	VAR robtarget Openhole_6212 := [[422.92, 1.19, 186.57], [-0.151917, 0.690595, 0.706732, 0.02301], [0,0,0,0], [9E9, 9E9, 9E9, 9E9, 9E9, 9E9]];
	VAR robtarget Openhole_6213 := [[423.41, 1.3, 186.5], [-0.15063, 0.690877, 0.706788, 0.021231], [0,0,0,0], [9E9, 9E9, 9E9, 9E9, 9E9, 9E9]];
	VAR robtarget Openhole_6214 := [[417.57, 1.3, 187.64], [-0.167714, 0.686929, 0.705941, 0.040584], [0,0,0,0], [9E9, 9E9, 9E9, 9E9, 9E9, 9E9]];
	VAR robtarget Openhole_6215 := [[417.07, 1.15, 187.69], [-0.168902, 0.686638, 0.705835, 0.042396], [0,0,0,0], [9E9, 9E9, 9E9, 9E9, 9E9, 9E9]];
	VAR robtarget Openhole_6216 := [[408.73, 0.11, 188.91], [-0.188817, 0.681431, 0.703403, 0.072276], [0,0,0,0], [9E9, 9E9, 9E9, 9E9, 9E9, 9E9]];
	VAR robtarget Openhole_6217 := [[397.88, -0.81, 190.45], [-0.213744, 0.674028, 0.698859, 0.107688], [0,0,0,0], [9E9, 9E9, 9E9, 9E9, 9E9, 9E9]];
	VAR robtarget Openhole_6218 := [[394.38, -1.04, 190.94], [-0.221411, 0.671548, 0.697131, 0.118354], [0,0,0,0], [9E9, 9E9, 9E9, 9E9, 9E9, 9E9]];
	VAR robtarget Openhole_6219 := [[389.38, -1.04, 191.81], [-0.232781, 0.667692, 0.694645, 0.13217], [0,0,0,0], [9E9, 9E9, 9E9, 9E9, 9E9, 9E9]];
	VAR robtarget Openhole_6220 := [[362.42, -1.04, 191.89], [-0.183051, 0.683002, 0.683002, 0.183051], [0,0,0,0], [9E9, 9E9, 9E9, 9E9, 9E9, 9E9]];
	VAR robtarget Openhole_6221 := [[362.42, -1.04, 192.01], [-0.183051, 0.683002, 0.683002, 0.183051], [0,0,0,0], [9E9, 9E9, 9E9, 9E9, 9E9, 9E9]];
	VAR robtarget Openhole_6222 := [[389.38, -1.04, 191.93], [-0.232953, 0.667632, 0.694664, 0.132066], [0,0,0,0], [9E9, 9E9, 9E9, 9E9, 9E9, 9E9]];
	VAR robtarget Openhole_6223 := [[394.38, -1.04, 191.06], [-0.221583, 0.671492, 0.697148, 0.118257], [0,0,0,0], [9E9, 9E9, 9E9, 9E9, 9E9, 9E9]];
	VAR robtarget Openhole_6224 := [[406.26, -0.14, 189.38], [-0.194769, 0.679754, 0.702502, 0.080567], [0,0,0,0], [9E9, 9E9, 9E9, 9E9, 9E9, 9E9]];
	VAR robtarget Openhole_6225 := [[415.12, 0.87, 188.1], [-0.173761, 0.685425, 0.705366, 0.049587], [0,0,0,0], [9E9, 9E9, 9E9, 9E9, 9E9, 9E9]];
	VAR robtarget Openhole_6226 := [[417.07, 1.15, 187.81], [-0.16906, 0.686599, 0.705837, 0.042358], [0,0,0,0], [9E9, 9E9, 9E9, 9E9, 9E9, 9E9]];
	VAR robtarget Openhole_6227 := [[417.57, 1.3, 187.76], [-0.167777, 0.686914, 0.705937, 0.040655], [0,0,0,0], [9E9, 9E9, 9E9, 9E9, 9E9, 9E9]];
	VAR robtarget Openhole_6228 := [[423.41, 1.3, 186.62], [-0.150696, 0.690862, 0.706786, 0.021304], [0,0,0,0], [9E9, 9E9, 9E9, 9E9, 9E9, 9E9]];
	VAR robtarget Openhole_6229 := [[422.92, 1.19, 186.69], [-0.152065, 0.690562, 0.706733, 0.02299], [0,0,0,0], [9E9, 9E9, 9E9, 9E9, 9E9, 9E9]];
	VAR robtarget Openhole_6230 := [[416.08, 0.05, 187.65], [-0.168515, 0.686733, 0.705405, 0.049029], [0,0,0,0], [9E9, 9E9, 9E9, 9E9, 9E9, 9E9]];
	VAR robtarget Openhole_6231 := [[407.72, -0.93, 188.8], [-0.188593, 0.681493, 0.702735, 0.078506], [0,0,0,0], [9E9, 9E9, 9E9, 9E9, 9E9, 9E9]];
	VAR robtarget Openhole_6232 := [[395.86, -1.84, 190.4], [-0.215851, 0.673356, 0.697466, 0.116368], [0,0,0,0], [9E9, 9E9, 9E9, 9E9, 9E9, 9E9]];
	VAR robtarget Openhole_6233 := [[394.38, -1.93, 190.59], [-0.219087, 0.67231, 0.696705, 0.120837], [0,0,0,0], [9E9, 9E9, 9E9, 9E9, 9E9, 9E9]];
	VAR robtarget Openhole_6234 := [[389.38, -1.93, 191.41], [-0.23052, 0.668476, 0.69418, 0.134588], [0,0,0,0], [9E9, 9E9, 9E9, 9E9, 9E9, 9E9]];
	VAR robtarget Openhole_6235 := [[362.38, -1.93, 191.5], [-0.183051, 0.683002, 0.683002, 0.183051], [0,0,0,0], [9E9, 9E9, 9E9, 9E9, 9E9, 9E9]];
	VAR robtarget Openhole_6236 := [[362.38, -2.82, 190.99], [-0.183051, 0.683002, 0.683002, 0.183051], [0,0,0,0], [9E9, 9E9, 9E9, 9E9, 9E9, 9E9]];
	VAR robtarget Openhole_6237 := [[374.38, -2.82, 190.95], [-0.183051, 0.683002, 0.683002, 0.183051], [0,0,0,0], [9E9, 9E9, 9E9, 9E9, 9E9, 9E9]];
	VAR robtarget Openhole_6238 := [[389.38, -2.82, 190.9], [-0.228098, 0.669306, 0.69369, 0.137092], [0,0,0,0], [9E9, 9E9, 9E9, 9E9, 9E9, 9E9]];
	VAR robtarget Openhole_6239 := [[394.37, -2.82, 190.12], [-0.21661, 0.673112, 0.696255, 0.123408], [0,0,0,0], [9E9, 9E9, 9E9, 9E9, 9E9, 9E9]];
	VAR robtarget Openhole_6240 := [[408.22, -1.78, 188.37], [-0.184687, 0.682562, 0.702618, 0.079551], [0,0,0,0], [9E9, 9E9, 9E9, 9E9, 9E9, 9E9]];
	VAR robtarget Openhole_6241 := [[416.11, -0.88, 187.35], [-0.165576, 0.687448, 0.705202, 0.05187], [0,0,0,0], [9E9, 9E9, 9E9, 9E9, 9E9, 9E9]];
	VAR robtarget Openhole_6242 := [[422.96, 0.24, 186.44], [-0.148993, 0.691232, 0.706633, 0.025886], [0,0,0,0], [9E9, 9E9, 9E9, 9E9, 9E9, 9E9]];
	VAR robtarget Openhole_6243 := [[427.32, 1.15, 185.82], [-0.138588, 0.693393, 0.707057, 0.008368], [0,0,0,0], [9E9, 9E9, 9E9, 9E9, 9E9, 9E9]];
	VAR robtarget Openhole_6244 := [[427.8, 1.3, 185.76], [-0.137346, 0.69364, 0.707077, 0.006493], [0,0,0,0], [9E9, 9E9, 9E9, 9E9, 9E9, 9E9]];
	VAR robtarget Openhole_6245 := [[431.7, 1.3, 185], [-0.125184, 0.695937, 0.707074, -0.006768], [0,0,0,0], [9E9, 9E9, 9E9, 9E9, 9E9, 9E9]];
	VAR robtarget Openhole_6246 := [[431.22, 1.07, 185.05], [-0.126171, 0.695759, 0.707092, -0.004584], [0,0,0,0], [9E9, 9E9, 9E9, 9E9, 9E9, 9E9]];
	VAR robtarget Openhole_6247 := [[423.97, -0.54, 186.06], [-0.143494, 0.692394, 0.706664, 0.025018], [0,0,0,0], [9E9, 9E9, 9E9, 9E9, 9E9, 9E9]];
	VAR robtarget Openhole_6248 := [[417.11, -1.69, 186.92], [-0.160194, 0.688722, 0.705255, 0.051147], [0,0,0,0], [9E9, 9E9, 9E9, 9E9, 9E9, 9E9]];
	VAR robtarget Openhole_6249 := [[409.23, -2.6, 187.89], [-0.179528, 0.683937, 0.702684, 0.078962], [0,0,0,0], [9E9, 9E9, 9E9, 9E9, 9E9, 9E9]];
	VAR robtarget Openhole_6250 := [[394.87, -3.67, 189.6], [-0.213029, 0.674254, 0.696063, 0.124485], [0,0,0,0], [9E9, 9E9, 9E9, 9E9, 9E9, 9E9]];
	VAR robtarget Openhole_6251 := [[394.37, -3.7, 189.65], [-0.214125, 0.673907, 0.695793, 0.125983], [0,0,0,0], [9E9, 9E9, 9E9, 9E9, 9E9, 9E9]];
	VAR robtarget Openhole_6252 := [[389.37, -3.7, 190.39], [-0.225669, 0.670129, 0.69319, 0.1396], [0,0,0,0], [9E9, 9E9, 9E9, 9E9, 9E9, 9E9]];
	VAR robtarget Openhole_6253 := [[362.37, -3.7, 190.48], [-0.183051, 0.683002, 0.683002, 0.183051], [0,0,0,0], [9E9, 9E9, 9E9, 9E9, 9E9, 9E9]];
	VAR robtarget Openhole_6254 := [[362.37, -4.58, 189.97], [-0.183051, 0.683002, 0.683002, 0.183051], [0,0,0,0], [9E9, 9E9, 9E9, 9E9, 9E9, 9E9]];
	VAR robtarget Openhole_6255 := [[374.37, -4.58, 189.93], [-0.183051, 0.683002, 0.683002, 0.183051], [0,0,0,0], [9E9, 9E9, 9E9, 9E9, 9E9, 9E9]];
	VAR robtarget Openhole_6256 := [[389.37, -4.59, 189.88], [-0.223232, 0.670945, 0.692679, 0.142111], [0,0,0,0], [9E9, 9E9, 9E9, 9E9, 9E9, 9E9]];
	VAR robtarget Openhole_6257 := [[394.36, -4.59, 189.19], [-0.211638, 0.674692, 0.69532, 0.128569], [0,0,0,0], [9E9, 9E9, 9E9, 9E9, 9E9, 9E9]];
	VAR robtarget Openhole_6258 := [[409.74, -3.48, 187.47], [-0.175466, 0.68499, 0.702554, 0.080113], [0,0,0,0], [9E9, 9E9, 9E9, 9E9, 9E9, 9E9]];
	VAR robtarget Openhole_6259 := [[417.63, -2.6, 186.56], [-0.155846, 0.689719, 0.705166, 0.052359], [0,0,0,0], [9E9, 9E9, 9E9, 9E9, 9E9, 9E9]];
	VAR robtarget Openhole_6260 := [[424, -1.56, 185.8], [-0.140137, 0.693081, 0.706546, 0.028167], [0,0,0,0], [9E9, 9E9, 9E9, 9E9, 9E9, 9E9]];
	VAR robtarget Openhole_6261 := [[430.79, -0.09, 184.92], [-0.123778, 0.696189, 0.707106, 0.000643], [0,0,0,0], [9E9, 9E9, 9E9, 9E9, 9E9, 9E9]];
	VAR robtarget Openhole_6262 := [[435.6, 1.08, 184.2], [-0.112198, 0.698149, 0.706837, -0.019526], [0,0,0,0], [9E9, 9E9, 9E9, 9E9, 9E9, 9E9]];
	VAR robtarget Openhole_6263 := [[436.08, 1.3, 184.14], [-0.111001, 0.69834, 0.706766, -0.021958], [0,0,0,0], [9E9, 9E9, 9E9, 9E9, 9E9, 9E9]];
	VAR robtarget Openhole_6264 := [[440.9, 1.3, 183.19], [-0.095242, 0.700663, 0.706058, -0.038495], [0,0,0,0], [9E9, 9E9, 9E9, 9E9, 9E9, 9E9]];
	VAR robtarget Openhole_6265 := [[440.43, 1.14, 183.27], [-0.096594, 0.700478, 0.706178, -0.03623], [0,0,0,0], [9E9, 9E9, 9E9, 9E9, 9E9, 9E9]];
	VAR robtarget Openhole_6266 := [[431.79, -1.04, 184.58], [-0.117568, 0.697265, 0.707107, 0.000299], [0,0,0,0], [9E9, 9E9, 9E9, 9E9, 9E9, 9E9]];
	VAR robtarget Openhole_6267 := [[425, -2.5, 185.42], [-0.134117, 0.694271, 0.706557, 0.027869], [0,0,0,0], [9E9, 9E9, 9E9, 9E9, 9E9, 9E9]];
	VAR robtarget Openhole_6268 := [[418.62, -3.5, 186.14], [-0.150147, 0.690982, 0.705191, 0.052021], [0,0,0,0], [9E9, 9E9, 9E9, 9E9, 9E9, 9E9]];
	VAR robtarget Openhole_6269 := [[410.22, -4.4, 187.05], [-0.171369, 0.686027, 0.702401, 0.081442], [0,0,0,0], [9E9, 9E9, 9E9, 9E9, 9E9, 9E9]];
	VAR robtarget Openhole_6270 := [[394.37, -5.47, 188.72], [-0.209106, 0.675481, 0.694846, 0.131109], [0,0,0,0], [9E9, 9E9, 9E9, 9E9, 9E9, 9E9]];
	VAR robtarget Openhole_6271 := [[389.37, -5.47, 189.37], [-0.22079, 0.671753, 0.692159, 0.144623], [0,0,0,0], [9E9, 9E9, 9E9, 9E9, 9E9, 9E9]];
	VAR robtarget Openhole_6272 := [[362.37, -5.47, 189.46], [-0.183051, 0.683002, 0.683002, 0.183051], [0,0,0,0], [9E9, 9E9, 9E9, 9E9, 9E9, 9E9]];
	VAR robtarget Openhole_6273 := [[362.37, -6.37, 188.93], [-0.183051, 0.683002, 0.683002, 0.183051], [0,0,0,0], [9E9, 9E9, 9E9, 9E9, 9E9, 9E9]];
	VAR robtarget Openhole_6274 := [[374.37, -6.37, 188.9], [-0.183051, 0.683002, 0.683002, 0.183051], [0,0,0,0], [9E9, 9E9, 9E9, 9E9, 9E9, 9E9]];
	VAR robtarget Openhole_6275 := [[389.37, -6.37, 188.85], [-0.21828, 0.672572, 0.691616, 0.147199], [0,0,0,0], [9E9, 9E9, 9E9, 9E9, 9E9, 9E9]];
	VAR robtarget Openhole_6276 := [[394.35, -6.37, 188.24], [-0.206567, 0.676262, 0.694335, 0.133787], [0,0,0,0], [9E9, 9E9, 9E9, 9E9, 9E9, 9E9]];
	VAR robtarget Openhole_6277 := [[411.75, -5.23, 186.54], [-0.164547, 0.687695, 0.702646, 0.079304], [0,0,0,0], [9E9, 9E9, 9E9, 9E9, 9E9, 9E9]];
	VAR robtarget Openhole_6278 := [[420.16, -4.36, 185.66], [-0.142875, 0.692522, 0.705352, 0.049787], [0,0,0,0], [9E9, 9E9, 9E9, 9E9, 9E9, 9E9]];
	VAR robtarget Openhole_6279 := [[427.03, -3.3, 184.92], [-0.125272, 0.695922, 0.70671, 0.023676], [0,0,0,0], [9E9, 9E9, 9E9, 9E9, 9E9, 9E9]];
	VAR robtarget Openhole_6280 := [[432.87, -2.08, 184.23], [-0.110768, 0.698377, 0.707107, 0.000055], [0,0,0,0], [9E9, 9E9, 9E9, 9E9, 9E9, 9E9]];
	VAR robtarget Openhole_6281 := [[441.01, 0.05, 183.07], [-0.091101, 0.701214, 0.706256, -0.034673], [0,0,0,0], [9E9, 9E9, 9E9, 9E9, 9E9, 9E9]];
	VAR robtarget Openhole_6282 := [[444.81, 1.13, 182.42], [-0.081961, 0.702341, 0.705254, -0.051157], [0,0,0,0], [9E9, 9E9, 9E9, 9E9, 9E9, 9E9]];
	VAR robtarget Openhole_6283 := [[445.28, 1.3, 182.34], [-0.080875, 0.702467, 0.705097, -0.053269], [0,0,0,0], [9E9, 9E9, 9E9, 9E9, 9E9, 9E9]];
	VAR robtarget Openhole_6284 := [[492.93, 1.3, 173.01], [0.078403, 0.702747, 0.678324, -0.199693], [0,0,0,0], [9E9, 9E9, 9E9, 9E9, 9E9, 9E9]];
	VAR robtarget Openhole_6285 := [[497.82, 0.35, 172.5], [0.096043, 0.700554, 0.675427, -0.209279], [0,0,0,0], [9E9, 9E9, 9E9, 9E9, 9E9, 9E9]];
	VAR robtarget Openhole_6286 := [[502.17, -0.75, 172.24], [0.112029, 0.698176, 0.673078, -0.216717], [0,0,0,0], [9E9, 9E9, 9E9, 9E9, 9E9, 9E9]];
	VAR robtarget Openhole_6287 := [[503.61, -1.18, 172.21], [0.117389, 0.697295, 0.67237, -0.218903], [0,0,0,0], [9E9, 9E9, 9E9, 9E9, 9E9, 9E9]];
	VAR robtarget Openhole_6288 := [[504.32, -1.34, 172.18], [0.119865, 0.696873, 0.671974, -0.220115], [0,0,0,0], [9E9, 9E9, 9E9, 9E9, 9E9, 9E9]];
	VAR robtarget Openhole_6289 := [[509.32, -1.34, 171.33], [0.183051, 0.683002, 0.683002, -0.183051], [0,0,0,0], [9E9, 9E9, 9E9, 9E9, 9E9, 9E9]];
	VAR robtarget Openhole_6290 := [[536.31, -1.34, 171.24], [0.183051, 0.683002, 0.683002, -0.183051], [0,0,0,0], [9E9, 9E9, 9E9, 9E9, 9E9, 9E9]];
	VAR robtarget Openhole_6291 := [[536.32, -1.86, 171.55], [0.183051, 0.683002, 0.683002, -0.183051], [0,0,0,0], [9E9, 9E9, 9E9, 9E9, 9E9, 9E9]];
	VAR robtarget Openhole_6292 := [[509.32, -1.86, 171.63], [0.183051, 0.683002, 0.683002, -0.183051], [0,0,0,0], [9E9, 9E9, 9E9, 9E9, 9E9, 9E9]];
	VAR robtarget Openhole_6293 := [[504.32, -1.86, 172.46], [0.121395, 0.696608, 0.672454, -0.218646], [0,0,0,0], [9E9, 9E9, 9E9, 9E9, 9E9, 9E9]];
	VAR robtarget Openhole_6294 := [[503.45, -1.68, 172.5], [0.118397, 0.697124, 0.672944, -0.217131], [0,0,0,0], [9E9, 9E9, 9E9, 9E9, 9E9, 9E9]];
	VAR robtarget Openhole_6295 := [[502.98, -1.51, 172.5], [0.116581, 0.69743, 0.673158, -0.216468], [0,0,0,0], [9E9, 9E9, 9E9, 9E9, 9E9, 9E9]];
	VAR robtarget Openhole_6296 := [[498.64, -0.34, 172.67], [0.100548, 0.699922, 0.675418, -0.20931], [0,0,0,0], [9E9, 9E9, 9E9, 9E9, 9E9, 9E9]];
	VAR robtarget Openhole_6297 := [[493.76, 0.68, 173.11], [0.082837, 0.702238, 0.678231, -0.200005], [0,0,0,0], [9E9, 9E9, 9E9, 9E9, 9E9, 9E9]];
	VAR robtarget Openhole_6298 := [[490.83, 1.18, 173.47], [0.07224, 0.703407, 0.680018, -0.193843], [0,0,0,0], [9E9, 9E9, 9E9, 9E9, 9E9, 9E9]];
	VAR robtarget Openhole_6299 := [[490.33, 1.3, 173.52], [0.07032, 0.703601, 0.680285, -0.192906], [0,0,0,0], [9E9, 9E9, 9E9, 9E9, 9E9, 9E9]];
	VAR robtarget Openhole_6300 := [[480.37, 1.3, 175.47], [0.038288, 0.706069, 0.68749, -0.1654], [0,0,0,0], [9E9, 9E9, 9E9, 9E9, 9E9, 9E9]];
	VAR robtarget Openhole_6301 := [[486.27, 0.75, 174.51], [0.059128, 0.70463, 0.683728, -0.180323], [0,0,0,0], [9E9, 9E9, 9E9, 9E9, 9E9, 9E9]];
	VAR robtarget Openhole_6302 := [[492.16, -0.08, 173.73], [0.080181, 0.702546, 0.680077, -0.193637], [0,0,0,0], [9E9, 9E9, 9E9, 9E9, 9E9, 9E9]];
	VAR robtarget Openhole_6303 := [[497.54, -1.09, 173.22], [0.099523, 0.700068, 0.676913, -0.204423], [0,0,0,0], [9E9, 9E9, 9E9, 9E9, 9E9, 9E9]];
	VAR robtarget Openhole_6304 := [[502.87, -2.42, 172.98], [0.118916, 0.697036, 0.674059, -0.213647], [0,0,0,0], [9E9, 9E9, 9E9, 9E9, 9E9, 9E9]];
	VAR robtarget Openhole_6305 := [[503.83, -2.67, 172.96], [0.122383, 0.696436, 0.673553, -0.215236], [0,0,0,0], [9E9, 9E9, 9E9, 9E9, 9E9, 9E9]];
	VAR robtarget Openhole_6306 := [[504.4, -2.79, 172.93], [0.124334, 0.69609, 0.67323, -0.216245], [0,0,0,0], [9E9, 9E9, 9E9, 9E9, 9E9, 9E9]];
	VAR robtarget Openhole_6307 := [[509.32, -2.79, 172.17], [0.183051, 0.683002, 0.683002, -0.183051], [0,0,0,0], [9E9, 9E9, 9E9, 9E9, 9E9, 9E9]];
	VAR robtarget Openhole_6308 := [[536.32, -2.79, 172.08], [0.183051, 0.683002, 0.683002, -0.183051], [0,0,0,0], [9E9, 9E9, 9E9, 9E9, 9E9, 9E9]];
	VAR robtarget Openhole_6309 := [[536.32, -3.66, 172.58], [0.183051, 0.683002, 0.683002, -0.183051], [0,0,0,0], [9E9, 9E9, 9E9, 9E9, 9E9, 9E9]];
	VAR robtarget Openhole_6310 := [[509.32, -3.66, 172.67], [0.183051, 0.683002, 0.683002, -0.183051], [0,0,0,0], [9E9, 9E9, 9E9, 9E9, 9E9, 9E9]];
	VAR robtarget Openhole_6311 := [[504.32, -3.66, 173.41], [0.12664, 0.695674, 0.674075, -0.213596], [0,0,0,0], [9E9, 9E9, 9E9, 9E9, 9E9, 9E9]];
	VAR robtarget Openhole_6312 := [[503.61, -3.55, 173.45], [0.124315, 0.696093, 0.674503, -0.21224], [0,0,0,0], [9E9, 9E9, 9E9, 9E9, 9E9, 9E9]];
	VAR robtarget Openhole_6313 := [[496.78, -2.08, 173.8], [0.100233, 0.699967, 0.678334, -0.199656], [0,0,0,0], [9E9, 9E9, 9E9, 9E9, 9E9, 9E9]];
	VAR robtarget Openhole_6314 := [[490.89, -1.1, 174.37], [0.079383, 0.702637, 0.681857, -0.187272], [0,0,0,0], [9E9, 9E9, 9E9, 9E9, 9E9, 9E9]];
	VAR robtarget Openhole_6315 := [[484.49, -0.34, 175.22], [0.056846, 0.704818, 0.685848, -0.172081], [0,0,0,0], [9E9, 9E9, 9E9, 9E9, 9E9, 9E9]];
	VAR robtarget Openhole_6316 := [[478.08, 0.04, 176.26], [0.034733, 0.706253, 0.689935, -0.154887], [0,0,0,0], [9E9, 9E9, 9E9, 9E9, 9E9, 9E9]];
	VAR robtarget Openhole_6317 := [[475.62, 0.08, 176.71], [0.02643, 0.706613, 0.691506, -0.147712], [0,0,0,0], [9E9, 9E9, 9E9, 9E9, 9E9, 9E9]];
	VAR robtarget Openhole_6318 := [[475.13, 0.08, 176.8], [0.02479, 0.706672, 0.691821, -0.146234], [0,0,0,0], [9E9, 9E9, 9E9, 9E9, 9E9, 9E9]];
	VAR robtarget Openhole_6319 := [[468.75, -0.12, 178.01], [0.00393, 0.707096, 0.69579, -0.126002], [0,0,0,0], [9E9, 9E9, 9E9, 9E9, 9E9, 9E9]];
	VAR robtarget Openhole_6320 := [[461.39, -0.49, 179.39], [-0.020021, 0.706823, 0.699814, -0.101296], [0,0,0,0], [9E9, 9E9, 9E9, 9E9, 9E9, 9E9]];
	VAR robtarget Openhole_6321 := [[460.9, -0.5, 179.48], [-0.021687, 0.706774, 0.700047, -0.099671], [0,0,0,0], [9E9, 9E9, 9E9, 9E9, 9E9, 9E9]];
	VAR robtarget Openhole_6322 := [[459.91, -0.49, 179.66], [-0.025088, 0.706662, 0.700494, -0.096476], [0,0,0,0], [9E9, 9E9, 9E9, 9E9, 9E9, 9E9]];
	VAR robtarget Openhole_6323 := [[457.95, -0.41, 180], [-0.032126, 0.706377, 0.701319, -0.090283], [0,0,0,0], [9E9, 9E9, 9E9, 9E9, 9E9, 9E9]];
	VAR robtarget Openhole_6324 := [[456.96, -0.33, 180.17], [-0.035756, 0.706202, 0.701698, -0.087291], [0,0,0,0], [9E9, 9E9, 9E9, 9E9, 9E9, 9E9]];
	VAR robtarget Openhole_6325 := [[455.49, -0.16, 180.42], [-0.041344, 0.705897, 0.702224, -0.082958], [0,0,0,0], [9E9, 9E9, 9E9, 9E9, 9E9, 9E9]];
	VAR robtarget Openhole_6326 := [[454.52, -0.01, 180.59], [-0.045187, 0.705661, 0.702542, -0.080213], [0,0,0,0], [9E9, 9E9, 9E9, 9E9, 9E9, 9E9]];
	VAR robtarget Openhole_6327 := [[453.56, 0.19, 180.76], [-0.049153, 0.705396, 0.702831, -0.077642], [0,0,0,0], [9E9, 9E9, 9E9, 9E9, 9E9, 9E9]];
	VAR robtarget Openhole_6328 := [[453.08, 0.32, 180.85], [-0.05122, 0.705249, 0.702957, -0.076494], [0,0,0,0], [9E9, 9E9, 9E9, 9E9, 9E9, 9E9]];
	VAR robtarget Openhole_6329 := [[451.65, 0.69, 181.1], [-0.057308, 0.704781, 0.703342, -0.072869], [0,0,0,0], [9E9, 9E9, 9E9, 9E9, 9E9, 9E9]];
	VAR robtarget Openhole_6330 := [[451.17, 0.77, 181.19], [-0.059249, 0.70462, 0.70348, -0.071529], [0,0,0,0], [9E9, 9E9, 9E9, 9E9, 9E9, 9E9]];
	VAR robtarget Openhole_6331 := [[450.68, 0.85, 181.29], [-0.061142, 0.704458, 0.703621, -0.070123], [0,0,0,0], [9E9, 9E9, 9E9, 9E9, 9E9, 9E9]];
	VAR robtarget Openhole_6332 := [[450.19, 0.88, 181.38], [-0.062918, 0.704302, 0.703774, -0.068577], [0,0,0,0], [9E9, 9E9, 9E9, 9E9, 9E9, 9E9]];
	VAR robtarget Openhole_6333 := [[449.7, 0.9, 181.47], [-0.064666, 0.704144, 0.703926, -0.066997], [0,0,0,0], [9E9, 9E9, 9E9, 9E9, 9E9, 9E9]];
	VAR robtarget Openhole_6334 := [[449.21, 0.87, 181.57], [-0.066224, 0.703999, 0.704091, -0.065232], [0,0,0,0], [9E9, 9E9, 9E9, 9E9, 9E9, 9E9]];
	VAR robtarget Openhole_6335 := [[448.72, 0.81, 181.66], [-0.067701, 0.703858, 0.704259, -0.063401], [0,0,0,0], [9E9, 9E9, 9E9, 9E9, 9E9, 9E9]];
	VAR robtarget Openhole_6336 := [[447.76, 0.61, 181.84], [-0.070294, 0.703604, 0.704601, -0.059475], [0,0,0,0], [9E9, 9E9, 9E9, 9E9, 9E9, 9E9]];
	VAR robtarget Openhole_6337 := [[446.81, 0.36, 182.02], [-0.072697, 0.70336, 0.704931, -0.055424], [0,0,0,0], [9E9, 9E9, 9E9, 9E9, 9E9, 9E9]];
	VAR robtarget Openhole_6338 := [[438.73, -1.98, 183.28], [-0.091999, 0.701096, 0.706817, -0.020235], [0,0,0,0], [9E9, 9E9, 9E9, 9E9, 9E9, 9E9]];
	VAR robtarget Openhole_6339 := [[433.44, -3.29, 183.95], [-0.10498, 0.69927, 0.707104, 0.002105], [0,0,0,0], [9E9, 9E9, 9E9, 9E9, 9E9, 9E9]];
	VAR robtarget Openhole_6340 := [[427.09, -4.48, 184.66], [-0.121297, 0.696625, 0.706578, 0.027349], [0,0,0,0], [9E9, 9E9, 9E9, 9E9, 9E9, 9E9]];
	VAR robtarget Openhole_6341 := [[419.69, -5.48, 185.41], [-0.140734, 0.69296, 0.704975, 0.054865], [0,0,0,0], [9E9, 9E9, 9E9, 9E9, 9E9, 9E9]];
	VAR robtarget Openhole_6342 := [[409.78, -6.33, 186.38], [-0.16668, 0.687181, 0.701508, 0.088809], [0,0,0,0], [9E9, 9E9, 9E9, 9E9, 9E9, 9E9]];
	VAR robtarget Openhole_6343 := [[394.35, -7.26, 187.77], [-0.204053, 0.677025, 0.693832, 0.136373], [0,0,0,0], [9E9, 9E9, 9E9, 9E9, 9E9, 9E9]];
	VAR robtarget Openhole_6344 := [[389.37, -7.26, 188.34], [-0.215823, 0.673365, 0.691075, 0.149715], [0,0,0,0], [9E9, 9E9, 9E9, 9E9, 9E9, 9E9]];
	VAR robtarget Openhole_6345 := [[362.37, -7.26, 188.42], [-0.183051, 0.683002, 0.683002, 0.183051], [0,0,0,0], [9E9, 9E9, 9E9, 9E9, 9E9, 9E9]];
	VAR robtarget Openhole_6346 := [[362.37, -8.14, 187.91], [-0.183051, 0.683002, 0.683002, 0.183051], [0,0,0,0], [9E9, 9E9, 9E9, 9E9, 9E9, 9E9]];
	VAR robtarget Openhole_6347 := [[374.37, -8.14, 187.88], [-0.183051, 0.683002, 0.683002, 0.183051], [0,0,0,0], [9E9, 9E9, 9E9, 9E9, 9E9, 9E9]];
	VAR robtarget Openhole_6348 := [[389.37, -8.14, 187.83], [-0.21336, 0.674149, 0.690525, 0.152233], [0,0,0,0], [9E9, 9E9, 9E9, 9E9, 9E9, 9E9]];
	VAR robtarget Openhole_6349 := [[394.35, -8.14, 187.31], [-0.201517, 0.677784, 0.693322, 0.13894], [0,0,0,0], [9E9, 9E9, 9E9, 9E9, 9E9, 9E9]];
	VAR robtarget Openhole_6350 := [[411.28, -7.19, 185.88], [-0.159838, 0.688805, 0.701751, 0.086865], [0,0,0,0], [9E9, 9E9, 9E9, 9E9, 9E9, 9E9]];
	VAR robtarget Openhole_6351 := [[421.2, -6.39, 184.97], [-0.133276, 0.694433, 0.705125, 0.052899], [0,0,0,0], [9E9, 9E9, 9E9, 9E9, 9E9, 9E9]];
	VAR robtarget Openhole_6352 := [[429.6, -5.33, 184.15], [-0.110628, 0.698399, 0.706773, 0.021733], [0,0,0,0], [9E9, 9E9, 9E9, 9E9, 9E9, 9E9]];
	VAR robtarget Openhole_6353 := [[435.95, -4.17, 183.46], [-0.093933, 0.70084, 0.707098, -0.003557], [0,0,0,0], [9E9, 9E9, 9E9, 9E9, 9E9, 9E9]];
	VAR robtarget Openhole_6354 := [[441.25, -2.83, 182.8], [-0.080832, 0.702472, 0.706629, -0.025984], [0,0,0,0], [9E9, 9E9, 9E9, 9E9, 9E9, 9E9]];
	VAR robtarget Openhole_6355 := [[446.48, -1.34, 182.03], [-0.06819, 0.703811, 0.705424, -0.048751], [0,0,0,0], [9E9, 9E9, 9E9, 9E9, 9E9, 9E9]];
	VAR robtarget Openhole_6356 := [[447.44, -1.11, 181.87], [-0.065687, 0.704049, 0.705136, -0.05276], [0,0,0,0], [9E9, 9E9, 9E9, 9E9, 9E9, 9E9]];
	VAR robtarget Openhole_6357 := [[447.93, -1.01, 181.79], [-0.064392, 0.704169, 0.704985, -0.054737], [0,0,0,0], [9E9, 9E9, 9E9, 9E9, 9E9, 9E9]];
	VAR robtarget Openhole_6358 := [[448.41, -0.92, 181.7], [-0.063039, 0.704291, 0.704832, -0.056671], [0,0,0,0], [9E9, 9E9, 9E9, 9E9, 9E9, 9E9]];
	VAR robtarget Openhole_6359 := [[448.9, -0.86, 181.62], [-0.061596, 0.704419, 0.704679, -0.058542], [0,0,0,0], [9E9, 9E9, 9E9, 9E9, 9E9, 9E9]];
	VAR robtarget Openhole_6360 := [[449.39, -0.83, 181.53], [-0.06, 0.704557, 0.704533, -0.060281], [0,0,0,0], [9E9, 9E9, 9E9, 9E9, 9E9, 9E9]];
	VAR robtarget Openhole_6361 := [[449.88, -0.83, 181.45], [-0.05834, 0.704696, 0.704387, -0.061965], [0,0,0,0], [9E9, 9E9, 9E9, 9E9, 9E9, 9E9]];
	VAR robtarget Openhole_6362 := [[450.38, -0.87, 181.36], [-0.05654, 0.704843, 0.70425, -0.0635], [0,0,0,0], [9E9, 9E9, 9E9, 9E9, 9E9, 9E9]];
	VAR robtarget Openhole_6363 := [[450.87, -0.92, 181.28], [-0.054694, 0.704988, 0.704115, -0.064977], [0,0,0,0], [9E9, 9E9, 9E9, 9E9, 9E9, 9E9]];
	VAR robtarget Openhole_6364 := [[451.35, -1, 181.19], [-0.052767, 0.705135, 0.703987, -0.066353], [0,0,0,0], [9E9, 9E9, 9E9, 9E9, 9E9, 9E9]];
	VAR robtarget Openhole_6365 := [[452.32, -1.2, 181.03], [-0.048803, 0.705421, 0.703738, -0.068943], [0,0,0,0], [9E9, 9E9, 9E9, 9E9, 9E9, 9E9]];
	VAR robtarget Openhole_6366 := [[452.8, -1.31, 180.95], [-0.046787, 0.705557, 0.703615, -0.070189], [0,0,0,0], [9E9, 9E9, 9E9, 9E9, 9E9, 9E9]];
	VAR robtarget Openhole_6367 := [[455.22, -1.78, 180.57], [-0.036925, 0.706142, 0.702928, -0.07676], [0,0,0,0], [9E9, 9E9, 9E9, 9E9, 9E9, 9E9]];
	VAR robtarget Openhole_6368 := [[459.15, -2.25, 179.96], [-0.021914, 0.706767, 0.70158, -0.088233], [0,0,0,0], [9E9, 9E9, 9E9, 9E9, 9E9, 9E9]];
	VAR robtarget Openhole_6369 := [[459.64, -2.28, 179.88], [-0.020126, 0.70682, 0.701387, -0.089759], [0,0,0,0], [9E9, 9E9, 9E9, 9E9, 9E9, 9E9]];
	VAR robtarget Openhole_6370 := [[460.13, -2.3, 179.8], [-0.018366, 0.706868, 0.701186, -0.091313], [0,0,0,0], [9E9, 9E9, 9E9, 9E9, 9E9, 9E9]];
	VAR robtarget Openhole_6371 := [[461.12, -2.32, 179.65], [-0.014919, 0.706949, 0.700766, -0.094483], [0,0,0,0], [9E9, 9E9, 9E9, 9E9, 9E9, 9E9]];
	VAR robtarget Openhole_6372 := [[466.05, -2.11, 178.82], [0.001205, 0.707106, 0.698325, -0.111093], [0,0,0,0], [9E9, 9E9, 9E9, 9E9, 9E9, 9E9]];
	VAR robtarget Openhole_6373 := [[473.41, -1.61, 177.5], [0.024487, 0.706683, 0.693963, -0.135703], [0,0,0,0], [9E9, 9E9, 9E9, 9E9, 9E9, 9E9]];
	VAR robtarget Openhole_6374 := [[476.86, -1.55, 176.91], [0.035783, 0.706201, 0.691807, -0.146296], [0,0,0,0], [9E9, 9E9, 9E9, 9E9, 9E9, 9E9]];
	VAR robtarget Openhole_6375 := [[477.36, -1.55, 176.83], [0.037424, 0.706116, 0.691497, -0.147757], [0,0,0,0], [9E9, 9E9, 9E9, 9E9, 9E9, 9E9]];
	VAR robtarget Openhole_6376 := [[483.28, -1.79, 175.91], [0.0575, 0.704765, 0.687764, -0.164256], [0,0,0,0], [9E9, 9E9, 9E9, 9E9, 9E9, 9E9]];
	VAR robtarget Openhole_6377 := [[489.2, -2.35, 175.14], [0.078019, 0.702789, 0.684075, -0.179001], [0,0,0,0], [9E9, 9E9, 9E9, 9E9, 9E9, 9E9]];
	VAR robtarget Openhole_6378 := [[496.1, -3.34, 174.48], [0.102013, 0.699709, 0.6799, -0.194259], [0,0,0,0], [9E9, 9E9, 9E9, 9E9, 9E9, 9E9]];
	VAR robtarget Openhole_6379 := [[501.51, -4.28, 174.13], [0.120516, 0.696761, 0.676713, -0.205083], [0,0,0,0], [9E9, 9E9, 9E9, 9E9, 9E9, 9E9]];
	VAR robtarget Openhole_6380 := [[503.48, -4.58, 174.01], [0.126978, 0.695612, 0.675519, -0.208985], [0,0,0,0], [9E9, 9E9, 9E9, 9E9, 9E9, 9E9]];
	VAR robtarget Openhole_6381 := [[504.32, -4.67, 173.94], [0.129589, 0.695131, 0.67497, -0.210749], [0,0,0,0], [9E9, 9E9, 9E9, 9E9, 9E9, 9E9]];
	VAR robtarget Openhole_6382 := [[509.32, -4.67, 173.25], [0.183051, 0.683002, 0.683002, -0.183051], [0,0,0,0], [9E9, 9E9, 9E9, 9E9, 9E9, 9E9]];
	VAR robtarget Openhole_6383 := [[536.32, -4.67, 173.17], [0.183051, 0.683002, 0.683002, -0.183051], [0,0,0,0], [9E9, 9E9, 9E9, 9E9, 9E9, 9E9]];
	VAR robtarget Openhole_6384 := [[536.32, -5.62, 173.72], [0.183051, 0.683002, 0.683002, -0.183051], [0,0,0,0], [9E9, 9E9, 9E9, 9E9, 9E9, 9E9]];
	VAR robtarget Openhole_6385 := [[524.32, -5.62, 173.75], [0.183051, 0.683002, 0.683002, -0.183051], [0,0,0,0], [9E9, 9E9, 9E9, 9E9, 9E9, 9E9]];
	VAR robtarget Openhole_6386 := [[509.32, -5.62, 173.8], [0.183051, 0.683002, 0.683002, -0.183051], [0,0,0,0], [9E9, 9E9, 9E9, 9E9, 9E9, 9E9]];
	VAR robtarget Openhole_6387 := [[504.32, -5.62, 174.45], [0.132347, 0.694611, 0.67581, -0.208039], [0,0,0,0], [9E9, 9E9, 9E9, 9E9, 9E9, 9E9]];
	VAR robtarget Openhole_6388 := [[503.82, -5.61, 174.51], [0.130937, 0.694878, 0.676166, -0.206882], [0,0,0,0], [9E9, 9E9, 9E9, 9E9, 9E9, 9E9]];
	VAR robtarget Openhole_6389 := [[498.86, -5.11, 174.91], [0.115421, 0.697623, 0.679366, -0.196117], [0,0,0,0], [9E9, 9E9, 9E9, 9E9, 9E9, 9E9]];
	VAR robtarget Openhole_6390 := [[489.97, -3.94, 175.64], [0.085306, 0.701942, 0.684772, -0.176317], [0,0,0,0], [9E9, 9E9, 9E9, 9E9, 9E9, 9E9]];
	VAR robtarget Openhole_6391 := [[483.54, -3.35, 176.38], [0.063277, 0.70427, 0.688722, -0.160194], [0,0,0,0], [9E9, 9E9, 9E9, 9E9, 9E9, 9E9]];
	VAR robtarget Openhole_6392 := [[478.1, -3.15, 177.15], [0.044992, 0.705674, 0.692088, -0.144964], [0,0,0,0], [9E9, 9E9, 9E9, 9E9, 9E9, 9E9]];
	VAR robtarget Openhole_6393 := [[477.6, -3.15, 177.22], [0.043366, 0.705776, 0.692394, -0.143495], [0,0,0,0], [9E9, 9E9, 9E9, 9E9, 9E9, 9E9]];
	VAR robtarget Openhole_6394 := [[477.11, -3.15, 177.3], [0.041739, 0.705874, 0.692698, -0.142018], [0,0,0,0], [9E9, 9E9, 9E9, 9E9, 9E9, 9E9]];
	VAR robtarget Openhole_6395 := [[471.69, -3.36, 178.17], [0.024402, 0.706686, 0.696008, -0.124794], [0,0,0,0], [9E9, 9E9, 9E9, 9E9, 9E9, 9E9]];
	VAR robtarget Openhole_6396 := [[462.34, -4.17, 179.68], [-0.004624, 0.707092, 0.70104, -0.092426], [0,0,0,0], [9E9, 9E9, 9E9, 9E9, 9E9, 9E9]];
	VAR robtarget Openhole_6397 := [[459.87, -4.23, 180.04], [-0.01287, 0.70699, 0.702086, -0.084116], [0,0,0,0], [9E9, 9E9, 9E9, 9E9, 9E9, 9E9]];
	VAR robtarget Openhole_6398 := [[459.37, -4.22, 180.11], [-0.01459, 0.706956, 0.702277, -0.082508], [0,0,0,0], [9E9, 9E9, 9E9, 9E9, 9E9, 9E9]];
	VAR robtarget Openhole_6399 := [[458.38, -4.18, 180.25], [-0.018111, 0.706875, 0.702638, -0.079368], [0,0,0,0], [9E9, 9E9, 9E9, 9E9, 9E9, 9E9]];
	VAR robtarget Openhole_6400 := [[457.4, -4.11, 180.39], [-0.021745, 0.706772, 0.702974, -0.076339], [0,0,0,0], [9E9, 9E9, 9E9, 9E9, 9E9, 9E9]];
	VAR robtarget Openhole_6401 := [[452.98, -3.48, 181], [-0.038952, 0.706033, 0.704235, -0.063669], [0,0,0,0], [9E9, 9E9, 9E9, 9E9, 9E9, 9E9]];
	VAR robtarget Openhole_6402 := [[451.03, -3.16, 181.28], [-0.046685, 0.705564, 0.704713, -0.058137], [0,0,0,0], [9E9, 9E9, 9E9, 9E9, 9E9, 9E9]];
	VAR robtarget Openhole_6403 := [[450.54, -3.1, 181.36], [-0.048568, 0.705437, 0.704831, -0.05669], [0,0,0,0], [9E9, 9E9, 9E9, 9E9, 9E9, 9E9]];
	VAR robtarget Openhole_6404 := [[449.56, -3.01, 181.51], [-0.052226, 0.705175, 0.705068, -0.053661], [0,0,0,0], [9E9, 9E9, 9E9, 9E9, 9E9, 9E9]];
	VAR robtarget Openhole_6405 := [[449.06, -3, 181.59], [-0.053951, 0.705046, 0.70519, -0.052032], [0,0,0,0], [9E9, 9E9, 9E9, 9E9, 9E9, 9E9]];
	VAR robtarget Openhole_6406 := [[448.57, -3, 181.66], [-0.05562, 0.704916, 0.705312, -0.050346], [0,0,0,0], [9E9, 9E9, 9E9, 9E9, 9E9, 9E9]];
	VAR robtarget Openhole_6407 := [[448.07, -3.04, 181.74], [-0.057166, 0.704792, 0.705438, -0.048548], [0,0,0,0], [9E9, 9E9, 9E9, 9E9, 9E9, 9E9]];
	VAR robtarget Openhole_6408 := [[447.58, -3.09, 181.81], [-0.05868, 0.704668, 0.705562, -0.046721], [0,0,0,0], [9E9, 9E9, 9E9, 9E9, 9E9, 9E9]];
	VAR robtarget Openhole_6409 := [[447.09, -3.15, 181.89], [-0.060126, 0.704546, 0.705684, -0.044841], [0,0,0,0], [9E9, 9E9, 9E9, 9E9, 9E9, 9E9]];
	VAR robtarget Openhole_6410 := [[446.12, -3.31, 182.03], [-0.062909, 0.704303, 0.705917, -0.040998], [0,0,0,0], [9E9, 9E9, 9E9, 9E9, 9E9, 9E9]];
	VAR robtarget Openhole_6411 := [[437.9, -5.24, 183.06], [-0.083953, 0.702105, 0.707076, -0.006619], [0,0,0,0], [9E9, 9E9, 9E9, 9E9, 9E9, 9E9]];
	VAR robtarget Openhole_6412 := [[431.53, -6.32, 183.72], [-0.101195, 0.699828, 0.706865, 0.018508], [0,0,0,0], [9E9, 9E9, 9E9, 9E9, 9E9, 9E9]];
	VAR robtarget Openhole_6413 := [[423.12, -7.3, 184.5], [-0.124507, 0.696059, 0.705367, 0.049576], [0,0,0,0], [9E9, 9E9, 9E9, 9E9, 9E9, 9E9]];
	VAR robtarget Openhole_6414 := [[413.19, -8.06, 185.36], [-0.151693, 0.690644, 0.702138, 0.083682], [0,0,0,0], [9E9, 9E9, 9E9, 9E9, 9E9, 9E9]];
	VAR robtarget Openhole_6415 := [[394.36, -9.02, 186.84], [-0.198951, 0.678541, 0.692808, 0.141482], [0,0,0,0], [9E9, 9E9, 9E9, 9E9, 9E9, 9E9]];
	VAR robtarget Openhole_6416 := [[389.36, -9.02, 187.32], [-0.210892, 0.674926, 0.689965, 0.154752], [0,0,0,0], [9E9, 9E9, 9E9, 9E9, 9E9, 9E9]];
	VAR robtarget Openhole_6417 := [[362.36, -9.02, 187.4], [-0.183051, 0.683002, 0.683002, 0.183051], [0,0,0,0], [9E9, 9E9, 9E9, 9E9, 9E9, 9E9]];
	VAR robtarget Openhole_6418 := [[362.36, -10.02, 186.83], [-0.183051, 0.683002, 0.683002, 0.183051], [0,0,0,0], [9E9, 9E9, 9E9, 9E9, 9E9, 9E9]];
	VAR robtarget Openhole_6419 := [[389.36, -10.02, 186.74], [-0.208089, 0.675795, 0.689319, 0.157605], [0,0,0,0], [9E9, 9E9, 9E9, 9E9, 9E9, 9E9]];
	VAR robtarget Openhole_6420 := [[394.36, -10.02, 186.31], [-0.196076, 0.679378, 0.692205, 0.144404], [0,0,0,0], [9E9, 9E9, 9E9, 9E9, 9E9, 9E9]];
	VAR robtarget Openhole_6421 := [[406.83, -9.43, 185.47], [-0.165342, 0.687504, 0.698919, 0.107296], [0,0,0,0], [9E9, 9E9, 9E9, 9E9, 9E9, 9E9]];
	VAR robtarget Openhole_6422 := [[420.77, -8.72, 184.38], [-0.127152, 0.695581, 0.704399, 0.061819], [0,0,0,0], [9E9, 9E9, 9E9, 9E9, 9E9, 9E9]];
	VAR robtarget Openhole_6423 := [[431.69, -7.82, 183.45], [-0.095766, 0.700592, 0.706736, 0.022902], [0,0,0,0], [9E9, 9E9, 9E9, 9E9, 9E9, 9E9]];
	VAR robtarget Openhole_6424 := [[439.1, -6.9, 182.74], [-0.074494, 0.703172, 0.707088, -0.005173], [0,0,0,0], [9E9, 9E9, 9E9, 9E9, 9E9, 9E9]];
	VAR robtarget Openhole_6425 := [[445.46, -5.78, 182.04], [-0.056884, 0.704815, 0.706446, -0.030565], [0,0,0,0], [9E9, 9E9, 9E9, 9E9, 9E9, 9E9]];
	VAR robtarget Openhole_6426 := [[446.45, -5.65, 181.92], [-0.053973, 0.705044, 0.706273, -0.034334], [0,0,0,0], [9E9, 9E9, 9E9, 9E9, 9E9, 9E9]];
	VAR robtarget Openhole_6427 := [[446.94, -5.6, 181.85], [-0.052463, 0.705158, 0.706181, -0.036175], [0,0,0,0], [9E9, 9E9, 9E9, 9E9, 9E9, 9E9]];
	VAR robtarget Openhole_6428 := [[447.43, -5.56, 181.79], [-0.050908, 0.705272, 0.706086, -0.037979], [0,0,0,0], [9E9, 9E9, 9E9, 9E9, 9E9, 9E9]];
	VAR robtarget Openhole_6429 := [[447.93, -5.54, 181.73], [-0.049298, 0.705386, 0.70599, -0.039734], [0,0,0,0], [9E9, 9E9, 9E9, 9E9, 9E9, 9E9]];
	VAR robtarget Openhole_6430 := [[448.43, -5.54, 181.66], [-0.047623, 0.705501, 0.705892, -0.041427], [0,0,0,0], [9E9, 9E9, 9E9, 9E9, 9E9, 9E9]];
	VAR robtarget Openhole_6431 := [[448.92, -5.55, 181.6], [-0.045907, 0.705615, 0.705793, -0.04308], [0,0,0,0], [9E9, 9E9, 9E9, 9E9, 9E9, 9E9]];
	VAR robtarget Openhole_6432 := [[450.41, -5.64, 181.4], [-0.040552, 0.705943, 0.705488, -0.047818], [0,0,0,0], [9E9, 9E9, 9E9, 9E9, 9E9, 9E9]];
	VAR robtarget Openhole_6433 := [[456.83, -6.26, 180.62], [-0.016497, 0.706914, 0.703895, -0.067321], [0,0,0,0], [9E9, 9E9, 9E9, 9E9, 9E9, 9E9]];
	VAR robtarget Openhole_6434 := [[457.32, -6.28, 180.56], [-0.014717, 0.706954, 0.703743, -0.068893], [0,0,0,0], [9E9, 9E9, 9E9, 9E9, 9E9, 9E9]];
	VAR robtarget Openhole_6435 := [[457.82, -6.3, 180.5], [-0.012971, 0.706988, 0.703584, -0.070495], [0,0,0,0], [9E9, 9E9, 9E9, 9E9, 9E9, 9E9]];
	VAR robtarget Openhole_6436 := [[458.32, -6.3, 180.44], [-0.011267, 0.707017, 0.703417, -0.072139], [0,0,0,0], [9E9, 9E9, 9E9, 9E9, 9E9, 9E9]];
	VAR robtarget Openhole_6437 := [[458.81, -6.29, 180.38], [-0.009594, 0.707042, 0.703244, -0.073808], [0,0,0,0], [9E9, 9E9, 9E9, 9E9, 9E9, 9E9]];
	VAR robtarget Openhole_6438 := [[459.31, -6.28, 180.32], [-0.007926, 0.707062, 0.703067, -0.07548], [0,0,0,0], [9E9, 9E9, 9E9, 9E9, 9E9, 9E9]];
	VAR robtarget Openhole_6439 := [[460.3, -6.24, 180.19], [-0.004681, 0.707091, 0.702692, -0.078893], [0,0,0,0], [9E9, 9E9, 9E9, 9E9, 9E9, 9E9]];
	VAR robtarget Openhole_6440 := [[461.29, -6.17, 180.06], [-0.001533, 0.707105, 0.702292, -0.082376], [0,0,0,0], [9E9, 9E9, 9E9, 9E9, 9E9, 9E9]];
	VAR robtarget Openhole_6441 := [[463.75, -5.92, 179.72], [0.006012, 0.707081, 0.701192, -0.091266], [0,0,0,0], [9E9, 9E9, 9E9, 9E9, 9E9, 9E9]];
	VAR robtarget Openhole_6442 := [[472.09, -4.91, 178.45], [0.030811, 0.706435, 0.696658, -0.121111], [0,0,0,0], [9E9, 9E9, 9E9, 9E9, 9E9, 9E9]];
	VAR robtarget Openhole_6443 := [[477.03, -4.63, 177.7], [0.046254, 0.705592, 0.693689, -0.137098], [0,0,0,0], [9E9, 9E9, 9E9, 9E9, 9E9, 9E9]];
	VAR robtarget Openhole_6444 := [[478.51, -4.61, 177.49], [0.051056, 0.705261, 0.692783, -0.141602], [0,0,0,0], [9E9, 9E9, 9E9, 9E9, 9E9, 9E9]];
	VAR robtarget Openhole_6445 := [[479.01, -4.61, 177.42], [0.052671, 0.705142, 0.692481, -0.143072], [0,0,0,0], [9E9, 9E9, 9E9, 9E9, 9E9, 9E9]];
	VAR robtarget Openhole_6446 := [[484.46, -4.79, 176.73], [0.070766, 0.703557, 0.689142, -0.158376], [0,0,0,0], [9E9, 9E9, 9E9, 9E9, 9E9, 9E9]];
	VAR robtarget Openhole_6447 := [[491.4, -5.38, 176.02], [0.094142, 0.700812, 0.684895, -0.175836], [0,0,0,0], [9E9, 9E9, 9E9, 9E9, 9E9, 9E9]];
	VAR robtarget Openhole_6448 := [[500.82, -6.37, 175.27], [0.124755, 0.696014, 0.679005, -0.197364], [0,0,0,0], [9E9, 9E9, 9E9, 9E9, 9E9, 9E9]];
	VAR robtarget Openhole_6449 := [[503.8, -6.51, 174.98], [0.133501, 0.69439, 0.676955, -0.204285], [0,0,0,0], [9E9, 9E9, 9E9, 9E9, 9E9, 9E9]];
	VAR robtarget Openhole_6450 := [[504.3, -6.51, 174.92], [0.134871, 0.694125, 0.676592, -0.205482], [0,0,0,0], [9E9, 9E9, 9E9, 9E9, 9E9, 9E9]];
	VAR robtarget Openhole_6451 := [[504.33, -6.51, 174.91], [0.134957, 0.694108, 0.676572, -0.20555], [0,0,0,0], [9E9, 9E9, 9E9, 9E9, 9E9, 9E9]];
	VAR robtarget Openhole_6452 := [[509.32, -6.51, 174.31], [0.183051, 0.683002, 0.683002, -0.183051], [0,0,0,0], [9E9, 9E9, 9E9, 9E9, 9E9, 9E9]];
	VAR robtarget Openhole_6453 := [[536.32, -6.51, 174.23], [0.183051, 0.683002, 0.683002, -0.183051], [0,0,0,0], [9E9, 9E9, 9E9, 9E9, 9E9, 9E9]];
	VAR robtarget Openhole_6454 := [[536.33, -7.39, 174.74], [0.183051, 0.683002, 0.683002, -0.183051], [0,0,0,0], [9E9, 9E9, 9E9, 9E9, 9E9, 9E9]];
	VAR robtarget Openhole_6455 := [[509.33, -7.39, 174.82], [0.183051, 0.683002, 0.683002, -0.183051], [0,0,0,0], [9E9, 9E9, 9E9, 9E9, 9E9, 9E9]];
	VAR robtarget Openhole_6456 := [[504.33, -7.39, 175.38], [0.137544, 0.6936, 0.67733, -0.203037], [0,0,0,0], [9E9, 9E9, 9E9, 9E9, 9E9, 9E9]];
	VAR robtarget Openhole_6457 := [[503.78, -7.39, 175.44], [0.136036, 0.693898, 0.677721, -0.201728], [0,0,0,0], [9E9, 9E9, 9E9, 9E9, 9E9, 9E9]];
	VAR robtarget Openhole_6458 := [[499.31, -7.22, 175.86], [0.123024, 0.696323, 0.680801, -0.191075], [0,0,0,0], [9E9, 9E9, 9E9, 9E9, 9E9, 9E9]];
	VAR robtarget Openhole_6459 := [[487.39, -6.24, 176.86], [0.084517, 0.702038, 0.688255, -0.162188], [0,0,0,0], [9E9, 9E9, 9E9, 9E9, 9E9, 9E9]];
	VAR robtarget Openhole_6460 := [[481.43, -5.99, 177.51], [0.06491, 0.704121, 0.691892, -0.145896], [0,0,0,0], [9E9, 9E9, 9E9, 9E9, 9E9, 9E9]];
	VAR robtarget Openhole_6461 := [[479.94, -5.98, 177.7], [0.060092, 0.704549, 0.692797, -0.141536], [0,0,0,0], [9E9, 9E9, 9E9, 9E9, 9E9, 9E9]];
	VAR robtarget Openhole_6462 := [[479.45, -5.98, 177.76], [0.0585, 0.704683, 0.693098, -0.140054], [0,0,0,0], [9E9, 9E9, 9E9, 9E9, 9E9, 9E9]];
	VAR robtarget Openhole_6463 := [[474.99, -6.17, 178.37], [0.044555, 0.705702, 0.695789, -0.126008], [0,0,0,0], [9E9, 9E9, 9E9, 9E9, 9E9, 9E9]];
	VAR robtarget Openhole_6464 := [[470.08, -6.73, 179.09], [0.030081, 0.706467, 0.698673, -0.108887], [0,0,0,0], [9E9, 9E9, 9E9, 9E9, 9E9, 9E9]];
	VAR robtarget Openhole_6465 := [[463.75, -7.88, 180], [0.012533, 0.706996, 0.702005, -0.084787], [0,0,0,0], [9E9, 9E9, 9E9, 9E9, 9E9, 9E9]];
	VAR robtarget Openhole_6466 := [[456.91, -9.15, 180.82], [-0.006471, 0.707077, 0.704727, -0.057962], [0,0,0,0], [9E9, 9E9, 9E9, 9E9, 9E9, 9E9]];
	VAR robtarget Openhole_6467 := [[453.96, -9.56, 181.12], [-0.015215, 0.706943, 0.705564, -0.046682], [0,0,0,0], [9E9, 9E9, 9E9, 9E9, 9E9, 9E9]];
	VAR robtarget Openhole_6468 := [[453.46, -9.61, 181.17], [-0.01671, 0.706909, 0.705685, -0.044822], [0,0,0,0], [9E9, 9E9, 9E9, 9E9, 9E9, 9E9]];
	VAR robtarget Openhole_6469 := [[452.97, -9.66, 181.22], [-0.018248, 0.706871, 0.705798, -0.042995], [0,0,0,0], [9E9, 9E9, 9E9, 9E9, 9E9, 9E9]];
	VAR robtarget Openhole_6470 := [[451.48, -9.76, 181.35], [-0.023013, 0.706732, 0.706105, -0.037633], [0,0,0,0], [9E9, 9E9, 9E9, 9E9, 9E9, 9E9]];
	VAR robtarget Openhole_6471 := [[450.48, -9.77, 181.44], [-0.026371, 0.706615, 0.706278, -0.03422], [0,0,0,0], [9E9, 9E9, 9E9, 9E9, 9E9, 9E9]];
	VAR robtarget Openhole_6472 := [[447, -9.62, 181.75], [-0.038752, 0.706044, 0.706735, -0.022918], [0,0,0,0], [9E9, 9E9, 9E9, 9E9, 9E9, 9E9]];
	VAR robtarget Openhole_6473 := [[445.01, -9.52, 181.94], [-0.045844, 0.705619, 0.706914, -0.016498], [0,0,0,0], [9E9, 9E9, 9E9, 9E9, 9E9, 9E9]];
	VAR robtarget Openhole_6474 := [[443.51, -9.49, 182.08], [-0.050971, 0.705267, 0.707013, -0.011493], [0,0,0,0], [9E9, 9E9, 9E9, 9E9, 9E9, 9E9]];
	VAR robtarget Openhole_6475 := [[433.06, -9.93, 182.97], [-0.084291, 0.702065, 0.706653, 0.025316], [0,0,0,0], [9E9, 9E9, 9E9, 9E9, 9E9, 9E9]];
	VAR robtarget Openhole_6476 := [[412.14, -10.76, 184.5], [-0.146288, 0.691809, 0.700637, 0.095436], [0,0,0,0], [9E9, 9E9, 9E9, 9E9, 9E9, 9E9]];
	VAR robtarget Openhole_6477 := [[397.17, -11.31, 185.42], [-0.185299, 0.682396, 0.693001, 0.140532], [0,0,0,0], [9E9, 9E9, 9E9, 9E9, 9E9, 9E9]];
	VAR robtarget Openhole_6478 := [[394.36, -11.45, 185.55], [-0.191958, 0.680553, 0.691321, 0.14858], [0,0,0,0], [9E9, 9E9, 9E9, 9E9, 9E9, 9E9]];
	VAR robtarget Openhole_6479 := [[389.36, -11.45, 185.92], [-0.204076, 0.677018, 0.688374, 0.16168], [0,0,0,0], [9E9, 9E9, 9E9, 9E9, 9E9, 9E9]];
	VAR robtarget Openhole_6480 := [[360.28, -11.45, 186.01], [-0.183051, 0.683002, 0.683002, 0.183051], [0,0,0,0], [9E9, 9E9, 9E9, 9E9, 9E9, 9E9]];
	VAR robtarget Openhole_6481 := [[360.24, -35.51, 172.11], [-0.183051, 0.683002, 0.683002, 0.183051], [0,0,0,0], [9E9, 9E9, 9E9, 9E9, 9E9, 9E9]];
	VAR robtarget Openhole_6482 := [[389.32, -35.51, 172.02], [-0.135486, 0.694005, 0.668864, 0.229391], [0,0,0,0], [9E9, 9E9, 9E9, 9E9, 9E9, 9E9]];
	VAR robtarget Openhole_6483 := [[394.32, -35.51, 172.82], [-0.121645, 0.696565, 0.672662, 0.218003], [0,0,0,0], [9E9, 9E9, 9E9, 9E9, 9E9, 9E9]];
	VAR robtarget Openhole_6484 := [[394.71, -35.54, 172.86], [-0.12045, 0.696772, 0.672937, 0.217153], [0,0,0,0], [9E9, 9E9, 9E9, 9E9, 9E9, 9E9]];
	VAR robtarget Openhole_6485 := [[395.19, -35.69, 172.86], [-0.118648, 0.697081, 0.673157, 0.216471], [0,0,0,0], [9E9, 9E9, 9E9, 9E9, 9E9, 9E9]];
	VAR robtarget Openhole_6486 := [[399.53, -36.88, 172.98], [-0.102571, 0.699628, 0.675375, 0.209447], [0,0,0,0], [9E9, 9E9, 9E9, 9E9, 9E9, 9E9]];
	VAR robtarget Openhole_6487 := [[404.89, -38.02, 173.42], [-0.083009, 0.702218, 0.678432, 0.199325], [0,0,0,0], [9E9, 9E9, 9E9, 9E9, 9E9, 9E9]];
	VAR robtarget Openhole_6488 := [[408.32, -38.6, 173.82], [-0.070585, 0.703575, 0.680502, 0.192137], [0,0,0,0], [9E9, 9E9, 9E9, 9E9, 9E9, 9E9]];
	VAR robtarget Openhole_6489 := [[408.81, -38.7, 173.87], [-0.06874, 0.703758, 0.680787, 0.191127], [0,0,0,0], [9E9, 9E9, 9E9, 9E9, 9E9, 9E9]];
	VAR robtarget Openhole_6490 := [[419.28, -38.7, 175.85], [-0.034891, 0.706245, 0.688262, 0.162157], [0,0,0,0], [9E9, 9E9, 9E9, 9E9, 9E9, 9E9]];
	VAR robtarget Openhole_6491 := [[418.78, -38.66, 175.77], [-0.036656, 0.706156, 0.687958, 0.163446], [0,0,0,0], [9E9, 9E9, 9E9, 9E9, 9E9, 9E9]];
	VAR robtarget Openhole_6492 := [[412.88, -38.13, 174.84], [-0.057542, 0.704762, 0.684216, 0.178462], [0,0,0,0], [9E9, 9E9, 9E9, 9E9, 9E9, 9E9]];
	VAR robtarget Openhole_6493 := [[406.49, -37.23, 174.04], [-0.080476, 0.702512, 0.680298, 0.192861], [0,0,0,0], [9E9, 9E9, 9E9, 9E9, 9E9, 9E9]];
	VAR robtarget Openhole_6494 := [[401.11, -36.21, 173.57], [-0.099889, 0.700016, 0.677158, 0.20361], [0,0,0,0], [9E9, 9E9, 9E9, 9E9, 9E9, 9E9]];
	VAR robtarget Openhole_6495 := [[395.29, -34.79, 173.34], [-0.121013, 0.696675, 0.674039, 0.213708], [0,0,0,0], [9E9, 9E9, 9E9, 9E9, 9E9, 9E9]];
	VAR robtarget Openhole_6496 := [[394.24, -34.53, 173.32], [-0.124753, 0.696015, 0.673488, 0.215439], [0,0,0,0], [9E9, 9E9, 9E9, 9E9, 9E9, 9E9]];
	VAR robtarget Openhole_6497 := [[389.32, -34.53, 172.59], [-0.138284, 0.693453, 0.669782, 0.226699], [0,0,0,0], [9E9, 9E9, 9E9, 9E9, 9E9, 9E9]];
	VAR robtarget Openhole_6498 := [[362.32, -34.53, 172.67], [-0.183051, 0.683002, 0.683002, 0.183051], [0,0,0,0], [9E9, 9E9, 9E9, 9E9, 9E9, 9E9]];
	VAR robtarget Openhole_6499 := [[362.32, -33.65, 173.18], [-0.183051, 0.683002, 0.683002, 0.183051], [0,0,0,0], [9E9, 9E9, 9E9, 9E9, 9E9, 9E9]];
	VAR robtarget Openhole_6500 := [[389.32, -33.65, 173.09], [-0.14077, 0.692953, 0.670588, 0.224301], [0,0,0,0], [9E9, 9E9, 9E9, 9E9, 9E9, 9E9]];
	VAR robtarget Openhole_6501 := [[394.32, -33.65, 173.8], [-0.127055, 0.695598, 0.674332, 0.212784], [0,0,0,0], [9E9, 9E9, 9E9, 9E9, 9E9, 9E9]];
	VAR robtarget Openhole_6502 := [[395, -33.77, 173.83], [-0.124835, 0.696, 0.674736, 0.211499], [0,0,0,0], [9E9, 9E9, 9E9, 9E9, 9E9, 9E9]];
	VAR robtarget Openhole_6503 := [[402.33, -35.28, 174.19], [-0.099033, 0.700138, 0.678861, 0.197858], [0,0,0,0], [9E9, 9E9, 9E9, 9E9, 9E9, 9E9]];
	VAR robtarget Openhole_6504 := [[408.72, -36.33, 174.78], [-0.076329, 0.702975, 0.682662, 0.184315], [0,0,0,0], [9E9, 9E9, 9E9, 9E9, 9E9, 9E9]];
	VAR robtarget Openhole_6505 := [[414.63, -37, 175.54], [-0.05544, 0.70493, 0.686325, 0.170169], [0,0,0,0], [9E9, 9E9, 9E9, 9E9, 9E9, 9E9]];
	VAR robtarget Openhole_6506 := [[420.55, -37.36, 176.46], [-0.03494, 0.706243, 0.690066, 0.154303], [0,0,0,0], [9E9, 9E9, 9E9, 9E9, 9E9, 9E9]];
	VAR robtarget Openhole_6507 := [[424, -37.4, 177.06], [-0.023291, 0.706723, 0.692244, 0.144215], [0,0,0,0], [9E9, 9E9, 9E9, 9E9, 9E9, 9E9]];
	VAR robtarget Openhole_6508 := [[424.49, -37.4, 177.15], [-0.021653, 0.706775, 0.692554, 0.142719], [0,0,0,0], [9E9, 9E9, 9E9, 9E9, 9E9, 9E9]];
	VAR robtarget Openhole_6509 := [[431.37, -37.13, 178.41], [0.000777, 0.707106, 0.696738, 0.12065], [0,0,0,0], [9E9, 9E9, 9E9, 9E9, 9E9, 9E9]];
	VAR robtarget Openhole_6510 := [[437.27, -36.86, 179.47], [0.0201, 0.706821, 0.699868, 0.100917], [0,0,0,0], [9E9, 9E9, 9E9, 9E9, 9E9, 9E9]];
	VAR robtarget Openhole_6511 := [[437.76, -36.86, 179.55], [0.021787, 0.706771, 0.700098, 0.099311], [0,0,0,0], [9E9, 9E9, 9E9, 9E9, 9E9, 9E9]];
	VAR robtarget Openhole_6512 := [[438.25, -36.86, 179.64], [0.02348, 0.706717, 0.700324, 0.097705], [0,0,0,0], [9E9, 9E9, 9E9, 9E9, 9E9, 9E9]];
	VAR robtarget Openhole_6513 := [[442.19, -37.1, 180.3], [0.037764, 0.706098, 0.701915, 0.085527], [0,0,0,0], [9E9, 9E9, 9E9, 9E9, 9E9, 9E9]];
	VAR robtarget Openhole_6514 := [[443.17, -37.22, 180.46], [0.041529, 0.705886, 0.702256, 0.082683], [0,0,0,0], [9E9, 9E9, 9E9, 9E9, 9E9, 9E9]];
	VAR robtarget Openhole_6515 := [[444.14, -37.38, 180.62], [0.045396, 0.705648, 0.70257, 0.07997], [0,0,0,0], [9E9, 9E9, 9E9, 9E9, 9E9, 9E9]];
	VAR robtarget Openhole_6516 := [[445.11, -37.59, 180.78], [0.049377, 0.705381, 0.702856, 0.07742], [0,0,0,0], [9E9, 9E9, 9E9, 9E9, 9E9, 9E9]];
	VAR robtarget Openhole_6517 := [[446.06, -37.84, 180.95], [0.053468, 0.705082, 0.703113, 0.075051], [0,0,0,0], [9E9, 9E9, 9E9, 9E9, 9E9, 9E9]];
	VAR robtarget Openhole_6518 := [[447.02, -38.07, 181.12], [0.057482, 0.704766, 0.703374, 0.072564], [0,0,0,0], [9E9, 9E9, 9E9, 9E9, 9E9, 9E9]];
	VAR robtarget Openhole_6519 := [[447.51, -38.14, 181.2], [0.059395, 0.704608, 0.703514, 0.071186], [0,0,0,0], [9E9, 9E9, 9E9, 9E9, 9E9, 9E9]];
	VAR robtarget Openhole_6520 := [[448, -38.2, 181.29], [0.061258, 0.704448, 0.703659, 0.06974], [0,0,0,0], [9E9, 9E9, 9E9, 9E9, 9E9, 9E9]];
	VAR robtarget Openhole_6521 := [[448.49, -38.23, 181.38], [0.063008, 0.704294, 0.703814, 0.068165], [0,0,0,0], [9E9, 9E9, 9E9, 9E9, 9E9, 9E9]];
	VAR robtarget Openhole_6522 := [[448.98, -38.23, 181.47], [0.064685, 0.704142, 0.703972, 0.06651], [0,0,0,0], [9E9, 9E9, 9E9, 9E9, 9E9, 9E9]];
	VAR robtarget Openhole_6523 := [[449.47, -38.19, 181.56], [0.066204, 0.704001, 0.70414, 0.064711], [0,0,0,0], [9E9, 9E9, 9E9, 9E9, 9E9, 9E9]];
	VAR robtarget Openhole_6524 := [[449.96, -38.12, 181.65], [0.067638, 0.703864, 0.704308, 0.062847], [0,0,0,0], [9E9, 9E9, 9E9, 9E9, 9E9, 9E9]];
	VAR robtarget Openhole_6525 := [[450.91, -37.89, 181.83], [0.07014, 0.703619, 0.704653, 0.058861], [0,0,0,0], [9E9, 9E9, 9E9, 9E9, 9E9, 9E9]];
	VAR robtarget Openhole_6526 := [[459, -35.6, 183.08], [0.089662, 0.701399, 0.706707, 0.023789], [0,0,0,0], [9E9, 9E9, 9E9, 9E9, 9E9, 9E9]];
	VAR robtarget Openhole_6527 := [[464.29, -34.25, 183.73], [0.102525, 0.699635, 0.707106, 0.00132], [0,0,0,0], [9E9, 9E9, 9E9, 9E9, 9E9, 9E9]];
	VAR robtarget Openhole_6528 := [[471.13, -32.95, 184.46], [0.120059, 0.69684, 0.706629, -0.025988], [0,0,0,0], [9E9, 9E9, 9E9, 9E9, 9E9, 9E9]];
	VAR robtarget Openhole_6529 := [[479.03, -31.9, 185.22], [0.140781, 0.692951, 0.704933, -0.055399], [0,0,0,0], [9E9, 9E9, 9E9, 9E9, 9E9, 9E9]];
	VAR robtarget Openhole_6530 := [[488.95, -31.06, 186.13], [0.166653, 0.687188, 0.701433, -0.089399], [0,0,0,0], [9E9, 9E9, 9E9, 9E9, 9E9, 9E9]];
	VAR robtarget Openhole_6531 := [[504.38, -30.16, 187.44], [0.203906, 0.677069, 0.693705, -0.137016], [0,0,0,0], [9E9, 9E9, 9E9, 9E9, 9E9, 9E9]];
	VAR robtarget Openhole_6532 := [[509.37, -30.16, 187.97], [0.183051, 0.683002, 0.683002, -0.183051], [0,0,0,0], [9E9, 9E9, 9E9, 9E9, 9E9, 9E9]];
	VAR robtarget Openhole_6533 := [[536.37, -30.16, 187.89], [0.183051, 0.683002, 0.683002, -0.183051], [0,0,0,0], [9E9, 9E9, 9E9, 9E9, 9E9, 9E9]];
	VAR robtarget Openhole_6534 := [[536.37, -29.28, 187.38], [0.183051, 0.683002, 0.683002, -0.183051], [0,0,0,0], [9E9, 9E9, 9E9, 9E9, 9E9, 9E9]];
	VAR robtarget Openhole_6535 := [[509.37, -29.28, 187.46], [0.183051, 0.683002, 0.683002, -0.183051], [0,0,0,0], [9E9, 9E9, 9E9, 9E9, 9E9, 9E9]];
	VAR robtarget Openhole_6536 := [[504.36, -29.28, 186.97], [0.201352, 0.677833, 0.693198, -0.139558], [0,0,0,0], [9E9, 9E9, 9E9, 9E9, 9E9, 9E9]];
	VAR robtarget Openhole_6537 := [[485.08, -30.34, 185.43], [0.153555, 0.690232, 0.702607, -0.079647], [0,0,0,0], [9E9, 9E9, 9E9, 9E9, 9E9, 9E9]];
	VAR robtarget Openhole_6538 := [[476.14, -31.11, 184.66], [0.129602, 0.695128, 0.705438, -0.048553], [0,0,0,0], [9E9, 9E9, 9E9, 9E9, 9E9, 9E9]];
	VAR robtarget Openhole_6539 := [[468.24, -32.14, 183.93], [0.108302, 0.698764, 0.706852, -0.018984], [0,0,0,0], [9E9, 9E9, 9E9, 9E9, 9E9, 9E9]];
	VAR robtarget Openhole_6540 := [[461.89, -33.32, 183.27], [0.091631, 0.701145, 0.707078, 0.006414], [0,0,0,0], [9E9, 9E9, 9E9, 9E9, 9E9, 9E9]];
	VAR robtarget Openhole_6541 := [[456.12, -34.79, 182.57], [0.077414, 0.702856, 0.706428, 0.030973], [0,0,0,0], [9E9, 9E9, 9E9, 9E9, 9E9, 9E9]];
	VAR robtarget Openhole_6542 := [[451.33, -36.06, 181.87], [0.065524, 0.704064, 0.705233, 0.051443], [0,0,0,0], [9E9, 9E9, 9E9, 9E9, 9E9, 9E9]];
	VAR robtarget Openhole_6543 := [[450.85, -36.17, 181.79], [0.064231, 0.704183, 0.705086, 0.053422], [0,0,0,0], [9E9, 9E9, 9E9, 9E9, 9E9, 9E9]];
	VAR robtarget Openhole_6544 := [[449.88, -36.33, 181.63], [0.061481, 0.704429, 0.704784, 0.057265], [0,0,0,0], [9E9, 9E9, 9E9, 9E9, 9E9, 9E9]];
	VAR robtarget Openhole_6545 := [[449.38, -36.38, 181.55], [0.059981, 0.704558, 0.704634, 0.059089], [0,0,0,0], [9E9, 9E9, 9E9, 9E9, 9E9, 9E9]];
	VAR robtarget Openhole_6546 := [[448.89, -36.4, 181.47], [0.058354, 0.704695, 0.704488, 0.060804], [0,0,0,0], [9E9, 9E9, 9E9, 9E9, 9E9, 9E9]];
	VAR robtarget Openhole_6547 := [[448.4, -36.38, 181.38], [0.056626, 0.704836, 0.704346, 0.062419], [0,0,0,0], [9E9, 9E9, 9E9, 9E9, 9E9, 9E9]];
	VAR robtarget Openhole_6548 := [[447.91, -36.33, 181.3], [0.054796, 0.70498, 0.704212, 0.063916], [0,0,0,0], [9E9, 9E9, 9E9, 9E9, 9E9, 9E9]];
	VAR robtarget Openhole_6549 := [[447.42, -36.26, 181.22], [0.052887, 0.705126, 0.704084, 0.065317], [0,0,0,0], [9E9, 9E9, 9E9, 9E9, 9E9, 9E9]];
	VAR robtarget Openhole_6550 := [[446.93, -36.18, 181.14], [0.050948, 0.705269, 0.703956, 0.066675], [0,0,0,0], [9E9, 9E9, 9E9, 9E9, 9E9, 9E9]];
	VAR robtarget Openhole_6551 := [[442.57, -35.3, 180.48], [0.033111, 0.706331, 0.70275, 0.078375], [0,0,0,0], [9E9, 9E9, 9E9, 9E9, 9E9, 9E9]];
	VAR robtarget Openhole_6552 := [[440.11, -35, 180.12], [0.023714, 0.706709, 0.701914, 0.085538], [0,0,0,0], [9E9, 9E9, 9E9, 9E9, 9E9, 9E9]];
	VAR robtarget Openhole_6553 := [[439.13, -34.94, 179.98], [0.020113, 0.706821, 0.701538, 0.088572], [0,0,0,0], [9E9, 9E9, 9E9, 9E9, 9E9, 9E9]];
	VAR robtarget Openhole_6554 := [[437.15, -34.9, 179.68], [0.013198, 0.706984, 0.70071, 0.0949], [0,0,0,0], [9E9, 9E9, 9E9, 9E9, 9E9, 9E9]];
	VAR robtarget Openhole_6555 := [[436.66, -34.9, 179.6], [0.011524, 0.707013, 0.700487, 0.096527], [0,0,0,0], [9E9, 9E9, 9E9, 9E9, 9E9, 9E9]];
	VAR robtarget Openhole_6556 := [[431.24, -35.21, 178.72], [-0.005945, 0.707082, 0.697706, 0.114917], [0,0,0,0], [9E9, 9E9, 9E9, 9E9, 9E9, 9E9]];
	VAR robtarget Openhole_6557 := [[424.35, -35.64, 177.55], [-0.027808, 0.70656, 0.69359, 0.137598], [0,0,0,0], [9E9, 9E9, 9E9, 9E9, 9E9, 9E9]];
	VAR robtarget Openhole_6558 := [[421.88, -35.68, 177.14], [-0.035898, 0.706195, 0.692053, 0.145129], [0,0,0,0], [9E9, 9E9, 9E9, 9E9, 9E9, 9E9]];
	VAR robtarget Openhole_6559 := [[421.39, -35.68, 177.06], [-0.03754, 0.70611, 0.691745, 0.146591], [0,0,0,0], [9E9, 9E9, 9E9, 9E9, 9E9, 9E9]];
	VAR robtarget Openhole_6560 := [[415.95, -35.48, 176.26], [-0.055963, 0.704889, 0.688348, 0.161793], [0,0,0,0], [9E9, 9E9, 9E9, 9E9, 9E9, 9E9]];
	VAR robtarget Openhole_6561 := [[410.02, -34.94, 175.52], [-0.076531, 0.702953, 0.684682, 0.176664], [0,0,0,0], [9E9, 9E9, 9E9, 9E9, 9E9, 9E9]];
	VAR robtarget Openhole_6562 := [[403.61, -34.06, 174.93], [-0.098918, 0.700154, 0.680823, 0.190998], [0,0,0,0], [9E9, 9E9, 9E9, 9E9, 9E9, 9E9]];
	VAR robtarget Openhole_6563 := [[395.25, -32.64, 174.46], [-0.127441, 0.695528, 0.67591, 0.207715], [0,0,0,0], [9E9, 9E9, 9E9, 9E9, 9E9, 9E9]];
	VAR robtarget Openhole_6564 := [[394.32, -32.55, 174.38], [-0.13028, 0.695001, 0.675308, 0.209663], [0,0,0,0], [9E9, 9E9, 9E9, 9E9, 9E9, 9E9]];
	VAR robtarget Openhole_6565 := [[389.32, -32.55, 173.73], [-0.143919, 0.692306, 0.671599, 0.221258], [0,0,0,0], [9E9, 9E9, 9E9, 9E9, 9E9, 9E9]];
	VAR robtarget Openhole_6566 := [[362.32, -32.55, 173.82], [-0.183051, 0.683002, 0.683002, 0.183051], [0,0,0,0], [9E9, 9E9, 9E9, 9E9, 9E9, 9E9]];
	VAR robtarget Openhole_6567 := [[362.32, -31.54, 174.4], [-0.183051, 0.683002, 0.683002, 0.183051], [0,0,0,0], [9E9, 9E9, 9E9, 9E9, 9E9, 9E9]];
	VAR robtarget Openhole_6568 := [[374.32, -31.54, 174.36], [-0.183051, 0.683002, 0.683002, 0.183051], [0,0,0,0], [9E9, 9E9, 9E9, 9E9, 9E9, 9E9]];
	VAR robtarget Openhole_6569 := [[389.32, -31.54, 174.31], [-0.146793, 0.691702, 0.672509, 0.218475], [0,0,0,0], [9E9, 9E9, 9E9, 9E9, 9E9, 9E9]];
	VAR robtarget Openhole_6570 := [[394.33, -31.54, 174.92], [-0.133214, 0.694445, 0.67619, 0.206801], [0,0,0,0], [9E9, 9E9, 9E9, 9E9, 9E9, 9E9]];
	VAR robtarget Openhole_6571 := [[394.83, -31.57, 174.96], [-0.131748, 0.694725, 0.676528, 0.205693], [0,0,0,0], [9E9, 9E9, 9E9, 9E9, 9E9, 9E9]];
	VAR robtarget Openhole_6572 := [[399.78, -32.12, 175.3], [-0.116062, 0.697517, 0.679665, 0.195079], [0,0,0,0], [9E9, 9E9, 9E9, 9E9, 9E9, 9E9]];
	VAR robtarget Openhole_6573 := [[407.69, -33.18, 175.87], [-0.089226, 0.701455, 0.68442, 0.177676], [0,0,0,0], [9E9, 9E9, 9E9, 9E9, 9E9, 9E9]];
	VAR robtarget Openhole_6574 := [[414.62, -33.85, 176.59], [-0.065414, 0.704075, 0.688635, 0.160568], [0,0,0,0], [9E9, 9E9, 9E9, 9E9, 9E9, 9E9]];
	VAR robtarget Openhole_6575 := [[420.07, -34.09, 177.3], [-0.046999, 0.705543, 0.691969, 0.145529], [0,0,0,0], [9E9, 9E9, 9E9, 9E9, 9E9, 9E9]];
	VAR robtarget Openhole_6576 := [[421.06, -34.1, 177.44], [-0.043723, 0.705754, 0.692575, 0.142616], [0,0,0,0], [9E9, 9E9, 9E9, 9E9, 9E9, 9E9]];
	VAR robtarget Openhole_6577 := [[421.55, -34.1, 177.51], [-0.042094, 0.705853, 0.692878, 0.141138], [0,0,0,0], [9E9, 9E9, 9E9, 9E9, 9E9, 9E9]];
	VAR robtarget Openhole_6578 := [[426.98, -33.88, 178.35], [-0.024694, 0.706675, 0.69616, 0.123943], [0,0,0,0], [9E9, 9E9, 9E9, 9E9, 9E9, 9E9]];
	VAR robtarget Openhole_6579 := [[436.34, -33.07, 179.78], [0.004378, 0.707093, 0.701151, 0.091579], [0,0,0,0], [9E9, 9E9, 9E9, 9E9, 9E9, 9E9]];
	VAR robtarget Openhole_6580 := [[438.32, -33.02, 180.06], [0.010959, 0.707022, 0.701989, 0.084918], [0,0,0,0], [9E9, 9E9, 9E9, 9E9, 9E9, 9E9]];
	VAR robtarget Openhole_6581 := [[438.82, -33.02, 180.12], [0.012661, 0.706993, 0.702184, 0.083296], [0,0,0,0], [9E9, 9E9, 9E9, 9E9, 9E9, 9E9]];
	VAR robtarget Openhole_6582 := [[439.31, -33.03, 180.19], [0.014389, 0.70696, 0.702372, 0.081695], [0,0,0,0], [9E9, 9E9, 9E9, 9E9, 9E9, 9E9]];
	VAR robtarget Openhole_6583 := [[442.77, -33.27, 180.64], [0.027042, 0.70659, 0.703532, 0.07101], [0,0,0,0], [9E9, 9E9, 9E9, 9E9, 9E9, 9E9]];
	VAR robtarget Openhole_6584 := [[447.66, -34.06, 181.3], [0.046415, 0.705582, 0.704787, 0.057228], [0,0,0,0], [9E9, 9E9, 9E9, 9E9, 9E9, 9E9]];
	VAR robtarget Openhole_6585 := [[448.16, -34.12, 181.37], [0.048295, 0.705456, 0.704904, 0.055776], [0,0,0,0], [9E9, 9E9, 9E9, 9E9, 9E9, 9E9]];
	VAR robtarget Openhole_6586 := [[448.65, -34.17, 181.44], [0.050134, 0.705327, 0.705021, 0.054273], [0,0,0,0], [9E9, 9E9, 9E9, 9E9, 9E9, 9E9]];
	VAR robtarget Openhole_6587 := [[449.14, -34.2, 181.51], [0.05193, 0.705197, 0.705139, 0.052717], [0,0,0,0], [9E9, 9E9, 9E9, 9E9, 9E9, 9E9]];
	VAR robtarget Openhole_6588 := [[449.64, -34.22, 181.58], [0.053657, 0.705068, 0.705259, 0.05109], [0,0,0,0], [9E9, 9E9, 9E9, 9E9, 9E9, 9E9]];
	VAR robtarget Openhole_6589 := [[450.13, -34.22, 181.66], [0.05534, 0.704938, 0.705378, 0.049416], [0,0,0,0], [9E9, 9E9, 9E9, 9E9, 9E9, 9E9]];
	VAR robtarget Openhole_6590 := [[450.63, -34.2, 181.73], [0.056953, 0.704809, 0.705498, 0.047677], [0,0,0,0], [9E9, 9E9, 9E9, 9E9, 9E9, 9E9]];
	VAR robtarget Openhole_6591 := [[451.12, -34.17, 181.8], [0.058518, 0.704681, 0.705616, 0.045893], [0,0,0,0], [9E9, 9E9, 9E9, 9E9, 9E9, 9E9]];
	VAR robtarget Openhole_6592 := [[451.61, -34.11, 181.87], [0.060008, 0.704556, 0.705734, 0.044046], [0,0,0,0], [9E9, 9E9, 9E9, 9E9, 9E9, 9E9]];
	VAR robtarget Openhole_6593 := [[452.1, -34.05, 181.94], [0.061445, 0.704432, 0.705849, 0.042157], [0,0,0,0], [9E9, 9E9, 9E9, 9E9, 9E9, 9E9]];
	VAR robtarget Openhole_6594 := [[452.59, -33.96, 182.01], [0.062823, 0.70431, 0.705962, 0.040226], [0,0,0,0], [9E9, 9E9, 9E9, 9E9, 9E9, 9E9]];
	VAR robtarget Openhole_6595 := [[460.82, -32.06, 182.98], [0.083971, 0.702103, 0.707082, 0.005898], [0,0,0,0], [9E9, 9E9, 9E9, 9E9, 9E9, 9E9]];
	VAR robtarget Openhole_6596 := [[467.7, -30.95, 183.65], [0.102677, 0.699612, 0.706794, -0.021036], [0,0,0,0], [9E9, 9E9, 9E9, 9E9, 9E9, 9E9]];
	VAR robtarget Openhole_6597 := [[476.61, -29.98, 184.42], [0.127395, 0.695536, 0.705062, -0.053731], [0,0,0,0], [9E9, 9E9, 9E9, 9E9, 9E9, 9E9]];
	VAR robtarget Openhole_6598 := [[487.55, -29.21, 185.29], [0.157069, 0.689441, 0.701245, -0.090863], [0,0,0,0], [9E9, 9E9, 9E9, 9E9, 9E9, 9E9]];
	VAR robtarget Openhole_6599 := [[504.36, -28.38, 186.5], [0.198798, 0.678586, 0.69267, -0.142157], [0,0,0,0], [9E9, 9E9, 9E9, 9E9, 9E9, 9E9]];
	VAR robtarget Openhole_6600 := [[509.36, -28.38, 186.95], [0.183051, 0.683002, 0.683002, -0.183051], [0,0,0,0], [9E9, 9E9, 9E9, 9E9, 9E9, 9E9]];
	VAR robtarget Openhole_6601 := [[536.36, -28.38, 186.86], [0.183051, 0.683002, 0.683002, -0.183051], [0,0,0,0], [9E9, 9E9, 9E9, 9E9, 9E9, 9E9]];
	VAR robtarget Openhole_6602 := [[536.36, -27.26, 186.21], [0.183051, 0.683002, 0.683002, -0.183051], [0,0,0,0], [9E9, 9E9, 9E9, 9E9, 9E9, 9E9]];
	VAR robtarget Openhole_6603 := [[509.36, -27.26, 186.3], [0.183051, 0.683002, 0.683002, -0.183051], [0,0,0,0], [9E9, 9E9, 9E9, 9E9, 9E9, 9E9]];
	VAR robtarget Openhole_6604 := [[504.36, -27.26, 185.9], [0.195578, 0.679521, 0.691991, -0.145425], [0,0,0,0], [9E9, 9E9, 9E9, 9E9, 9E9, 9E9]];
	VAR robtarget Openhole_6605 := [[490.44, -27.87, 185.04], [0.161033, 0.688526, 0.699444, -0.10382], [0,0,0,0], [9E9, 9E9, 9E9, 9E9, 9E9, 9E9]];
	VAR robtarget Openhole_6606 := [[476.49, -28.59, 184.04], [0.122557, 0.696405, 0.704734, -0.057875], [0,0,0,0], [9E9, 9E9, 9E9, 9E9, 9E9, 9E9]];
	VAR robtarget Openhole_6607 := [[464.07, -29.6, 183.04], [0.086495, 0.701797, 0.706981, -0.013327], [0,0,0,0], [9E9, 9E9, 9E9, 9E9, 9E9, 9E9]];
	VAR robtarget Openhole_6608 := [[458.64, -30.3, 182.55], [0.070913, 0.703542, 0.707068, 0.007436], [0,0,0,0], [9E9, 9E9, 9E9, 9E9, 9E9, 9E9]];
	VAR robtarget Openhole_6609 := [[453.73, -31.11, 182.05], [0.057154, 0.704793, 0.706597, 0.026842], [0,0,0,0], [9E9, 9E9, 9E9, 9E9, 9E9, 9E9]];
	VAR robtarget Openhole_6610 := [[452.75, -31.23, 181.94], [0.054226, 0.705024, 0.706444, 0.030601], [0,0,0,0], [9E9, 9E9, 9E9, 9E9, 9E9, 9E9]];
	VAR robtarget Openhole_6611 := [[451.76, -31.32, 181.83], [0.051158, 0.705254, 0.706277, 0.034248], [0,0,0,0], [9E9, 9E9, 9E9, 9E9, 9E9, 9E9]];
	VAR robtarget Openhole_6612 := [[450.76, -31.35, 181.71], [0.047911, 0.705482, 0.706099, 0.037737], [0,0,0,0], [9E9, 9E9, 9E9, 9E9, 9E9, 9E9]];
	VAR robtarget Openhole_6613 := [[450.27, -31.35, 181.65], [0.046224, 0.705594, 0.706007, 0.03942], [0,0,0,0], [9E9, 9E9, 9E9, 9E9, 9E9, 9E9]];
	VAR robtarget Openhole_6614 := [[449.77, -31.34, 181.59], [0.044488, 0.705706, 0.705914, 0.041056], [0,0,0,0], [9E9, 9E9, 9E9, 9E9, 9E9, 9E9]];
	VAR robtarget Openhole_6615 := [[449.27, -31.31, 181.53], [0.042723, 0.705815, 0.705819, 0.042661], [0,0,0,0], [9E9, 9E9, 9E9, 9E9, 9E9, 9E9]];
	VAR robtarget Openhole_6616 := [[445.32, -30.96, 181.08], [0.028017, 0.706552, 0.704978, 0.054826], [0,0,0,0], [9E9, 9E9, 9E9, 9E9, 9E9, 9E9]];
	VAR robtarget Openhole_6617 := [[441.35, -30.75, 180.64], [0.013726, 0.706974, 0.703887, 0.067399], [0,0,0,0], [9E9, 9E9, 9E9, 9E9, 9E9, 9E9]];
	VAR robtarget Openhole_6618 := [[440.85, -30.75, 180.58], [0.012024, 0.707005, 0.703727, 0.06905], [0,0,0,0], [9E9, 9E9, 9E9, 9E9, 9E9, 9E9]];
	VAR robtarget Openhole_6619 := [[440.35, -30.75, 180.53], [0.010344, 0.707031, 0.703562, 0.070717], [0,0,0,0], [9E9, 9E9, 9E9, 9E9, 9E9, 9E9]];
	VAR robtarget Openhole_6620 := [[439.36, -30.78, 180.41], [0.00705, 0.707072, 0.703213, 0.074105], [0,0,0,0], [9E9, 9E9, 9E9, 9E9, 9E9, 9E9]];
	VAR robtarget Openhole_6621 := [[438.37, -30.84, 180.29], [0.003853, 0.707096, 0.70284, 0.077565], [0,0,0,0], [9E9, 9E9, 9E9, 9E9, 9E9, 9E9]];
	VAR robtarget Openhole_6622 := [[432.46, -31.52, 179.51], [-0.014003, 0.706968, 0.700139, 0.099019], [0,0,0,0], [9E9, 9E9, 9E9, 9E9, 9E9, 9E9]];
	VAR robtarget Openhole_6623 := [[426.07, -32.27, 178.58], [-0.033008, 0.706336, 0.696572, 0.121602], [0,0,0,0], [9E9, 9E9, 9E9, 9E9, 9E9, 9E9]];
	VAR robtarget Openhole_6624 := [[421.13, -32.53, 177.88], [-0.048556, 0.705438, 0.693619, 0.13745], [0,0,0,0], [9E9, 9E9, 9E9, 9E9, 9E9, 9E9]];
	VAR robtarget Openhole_6625 := [[419.64, -32.54, 177.68], [-0.053384, 0.705089, 0.69272, 0.141914], [0,0,0,0], [9E9, 9E9, 9E9, 9E9, 9E9, 9E9]];
	VAR robtarget Openhole_6626 := [[419.15, -32.54, 177.62], [-0.055007, 0.704964, 0.692419, 0.143373], [0,0,0,0], [9E9, 9E9, 9E9, 9E9, 9E9, 9E9]];
	VAR robtarget Openhole_6627 := [[413.19, -32.29, 176.93], [-0.074896, 0.703129, 0.688815, 0.159795], [0,0,0,0], [9E9, 9E9, 9E9, 9E9, 9E9, 9E9]];
	VAR robtarget Openhole_6628 := [[404.76, -31.51, 176.19], [-0.103269, 0.699525, 0.683694, 0.18045], [0,0,0,0], [9E9, 9E9, 9E9, 9E9, 9E9, 9E9]];
	VAR robtarget Openhole_6629 := [[397.32, -30.78, 175.66], [-0.127122, 0.695586, 0.679013, 0.197336], [0,0,0,0], [9E9, 9E9, 9E9, 9E9, 9E9, 9E9]];
	VAR robtarget Openhole_6630 := [[394.83, -30.66, 175.44], [-0.134407, 0.694215, 0.677313, 0.203095], [0,0,0,0], [9E9, 9E9, 9E9, 9E9, 9E9, 9E9]];
	VAR robtarget Openhole_6631 := [[389.33, -30.66, 174.82], [-0.149318, 0.691161, 0.673301, 0.216024], [0,0,0,0], [9E9, 9E9, 9E9, 9E9, 9E9, 9E9]];
	VAR robtarget Openhole_6632 := [[362.33, -30.66, 174.91], [-0.183051, 0.683002, 0.683002, 0.183051], [0,0,0,0], [9E9, 9E9, 9E9, 9E9, 9E9, 9E9]];
	VAR robtarget Openhole_6633 := [[362.33, -28.99, 175.87], [-0.183051, 0.683002, 0.683002, 0.183051], [0,0,0,0], [9E9, 9E9, 9E9, 9E9, 9E9, 9E9]];
	VAR robtarget Openhole_6634 := [[374.33, -28.99, 175.83], [-0.183051, 0.683002, 0.683002, 0.183051], [0,0,0,0], [9E9, 9E9, 9E9, 9E9, 9E9, 9E9]];
	VAR robtarget Openhole_6635 := [[389.33, -28.99, 175.79], [-0.154092, 0.690113, 0.674774, 0.211377], [0,0,0,0], [9E9, 9E9, 9E9, 9E9, 9E9, 9E9]];
	VAR robtarget Openhole_6636 := [[394.3, -28.99, 176.26], [-0.140772, 0.692953, 0.678354, 0.19959], [0,0,0,0], [9E9, 9E9, 9E9, 9E9, 9E9, 9E9]];
	VAR robtarget Openhole_6637 := [[394.83, -28.97, 176.33], [-0.139415, 0.693227, 0.678745, 0.198255], [0,0,0,0], [9E9, 9E9, 9E9, 9E9, 9E9, 9E9]];
	VAR robtarget Openhole_6638 := [[396.82, -28.94, 176.53], [-0.133987, 0.694296, 0.680177, 0.193284], [0,0,0,0], [9E9, 9E9, 9E9, 9E9, 9E9, 9E9]];
	VAR robtarget Openhole_6639 := [[397.31, -28.94, 176.58], [-0.132593, 0.694564, 0.680528, 0.192046], [0,0,0,0], [9E9, 9E9, 9E9, 9E9, 9E9, 9E9]];
	VAR robtarget Openhole_6640 := [[403.29, -29.19, 177.04], [-0.114712, 0.69774, 0.68448, 0.177448], [0,0,0,0], [9E9, 9E9, 9E9, 9E9, 9E9, 9E9]];
	VAR robtarget Openhole_6641 := [[414.24, -29.87, 177.88], [-0.079282, 0.702648, 0.691155, 0.149346], [0,0,0,0], [9E9, 9E9, 9E9, 9E9, 9E9, 9E9]];
	VAR robtarget Openhole_6642 := [[417.72, -29.94, 178.22], [-0.067981, 0.703831, 0.693224, 0.13943], [0,0,0,0], [9E9, 9E9, 9E9, 9E9, 9E9, 9E9]];
	VAR robtarget Openhole_6643 := [[418.21, -29.94, 178.27], [-0.066392, 0.703983, 0.693519, 0.137954], [0,0,0,0], [9E9, 9E9, 9E9, 9E9, 9E9, 9E9]];
	VAR robtarget Openhole_6644 := [[423.18, -29.75, 178.84], [-0.050855, 0.705276, 0.696428, 0.122423], [0,0,0,0], [9E9, 9E9, 9E9, 9E9, 9E9, 9E9]];
	VAR robtarget Openhole_6645 := [[427.61, -29.25, 179.4], [-0.037841, 0.706094, 0.698961, 0.10702], [0,0,0,0], [9E9, 9E9, 9E9, 9E9, 9E9, 9E9]];
	VAR robtarget Openhole_6646 := [[431.99, -28.38, 179.98], [-0.026029, 0.706628, 0.701324, 0.090251], [0,0,0,0], [9E9, 9E9, 9E9, 9E9, 9E9, 9E9]];
	VAR robtarget Openhole_6647 := [[436.77, -27.04, 180.57], [-0.014344, 0.706961, 0.70361, 0.070237], [0,0,0,0], [9E9, 9E9, 9E9, 9E9, 9E9, 9E9]];
	VAR robtarget Openhole_6648 := [[439.61, -26.14, 180.88], [-0.007714, 0.707065, 0.704741, 0.057798], [0,0,0,0], [9E9, 9E9, 9E9, 9E9, 9E9, 9E9]];
	VAR robtarget Openhole_6649 := [[441.02, -25.65, 181.01], [-0.004594, 0.707092, 0.705234, 0.051431], [0,0,0,0], [9E9, 9E9, 9E9, 9E9, 9E9, 9E9]];
	VAR robtarget Openhole_6650 := [[441.49, -25.47, 181.05], [-0.003615, 0.707098, 0.705388, 0.049275], [0,0,0,0], [9E9, 9E9, 9E9, 9E9, 9E9, 9E9]];
	VAR robtarget Openhole_6651 := [[441.94, -25.27, 181.1], [-0.002741, 0.707101, 0.705538, 0.047072], [0,0,0,0], [9E9, 9E9, 9E9, 9E9, 9E9, 9E9]];
	VAR robtarget Openhole_6652 := [[442.83, -24.81, 181.18], [-0.00127, 0.707106, 0.705825, 0.042561], [0,0,0,0], [9E9, 9E9, 9E9, 9E9, 9E9, 9E9]];
	VAR robtarget Openhole_6653 := [[443.59, -24.26, 181.25], [-0.000554, 0.707107, 0.706077, 0.038142], [0,0,0,0], [9E9, 9E9, 9E9, 9E9, 9E9, 9E9]];
	VAR robtarget Openhole_6654 := [[445.39, -24.26, 181.34], [0.005608, 0.707085, 0.70638, 0.032055], [0,0,0,0], [9E9, 9E9, 9E9, 9E9, 9E9, 9E9]];
	VAR robtarget Openhole_6655 := [[443.96, -22.2, 181.38], [-0.006288, 0.707079, 0.706472, 0.02996], [0,0,0,0], [9E9, 9E9, 9E9, 9E9, 9E9, 9E9]];
	VAR robtarget Openhole_6656 := [[442.15, -22.2, 181.32], [-0.012439, 0.706997, 0.706188, 0.036041], [0,0,0,0], [9E9, 9E9, 9E9, 9E9, 9E9, 9E9]];
	VAR robtarget Openhole_6657 := [[441.31, -22.66, 181.26], [-0.013735, 0.706973, 0.705951, 0.040418], [0,0,0,0], [9E9, 9E9, 9E9, 9E9, 9E9, 9E9]];
	VAR robtarget Openhole_6658 := [[440.05, -23.46, 181.14], [-0.015302, 0.706941, 0.70552, 0.04735], [0,0,0,0], [9E9, 9E9, 9E9, 9E9, 9E9, 9E9]];
	VAR robtarget Openhole_6659 := [[439.62, -23.72, 181.1], [-0.015888, 0.706928, 0.705362, 0.049639], [0,0,0,0], [9E9, 9E9, 9E9, 9E9, 9E9, 9E9]];
	VAR robtarget Openhole_6660 := [[438.31, -24.43, 180.97], [-0.017963, 0.706879, 0.704854, 0.056398], [0,0,0,0], [9E9, 9E9, 9E9, 9E9, 9E9, 9E9]];
	VAR robtarget Openhole_6661 := [[435.13, -25.85, 180.61], [-0.023933, 0.706702, 0.703468, 0.07164], [0,0,0,0], [9E9, 9E9, 9E9, 9E9, 9E9, 9E9]];
	VAR robtarget Openhole_6662 := [[434.67, -26.03, 180.55], [-0.024888, 0.706669, 0.703249, 0.07376], [0,0,0,0], [9E9, 9E9, 9E9, 9E9, 9E9, 9E9]];
	VAR robtarget Openhole_6663 := [[433.73, -26.37, 180.44], [-0.026886, 0.706595, 0.702798, 0.077944], [0,0,0,0], [9E9, 9E9, 9E9, 9E9, 9E9, 9E9]];
	VAR robtarget Openhole_6664 := [[432.32, -26.83, 180.26], [-0.030135, 0.706464, 0.702092, 0.084062], [0,0,0,0], [9E9, 9E9, 9E9, 9E9, 9E9, 9E9]];
	VAR robtarget Openhole_6665 := [[430.4, -27.35, 180.02], [-0.034823, 0.706249, 0.701102, 0.091956], [0,0,0,0], [9E9, 9E9, 9E9, 9E9, 9E9, 9E9]];
	VAR robtarget Openhole_6666 := [[427, -28.06, 179.6], [-0.043803, 0.705749, 0.699255, 0.10508], [0,0,0,0], [9E9, 9E9, 9E9, 9E9, 9E9, 9E9]];
	VAR robtarget Openhole_6667 := [[422.56, -28.57, 179.08], [-0.056758, 0.704825, 0.696764, 0.120501], [0,0,0,0], [9E9, 9E9, 9E9, 9E9, 9E9, 9E9]];
	VAR robtarget Openhole_6668 := [[417.09, -28.75, 178.52], [-0.073823, 0.703243, 0.693608, 0.137507], [0,0,0,0], [9E9, 9E9, 9E9, 9E9, 9E9, 9E9]];
	VAR robtarget Openhole_6669 := [[416.6, -28.75, 178.48], [-0.07541, 0.703074, 0.693316, 0.138969], [0,0,0,0], [9E9, 9E9, 9E9, 9E9, 9E9, 9E9]];
	VAR robtarget Openhole_6670 := [[408.63, -28.45, 177.85], [-0.10111, 0.699841, 0.688585, 0.16078], [0,0,0,0], [9E9, 9E9, 9E9, 9E9, 9E9, 9E9]];
	VAR robtarget Openhole_6671 := [[399.66, -28.03, 177.24], [-0.12871, 0.695294, 0.682895, 0.183453], [0,0,0,0], [9E9, 9E9, 9E9, 9E9, 9E9, 9E9]];
	VAR robtarget Openhole_6672 := [[398.16, -28.02, 177.11], [-0.132968, 0.694492, 0.681871, 0.187222], [0,0,0,0], [9E9, 9E9, 9E9, 9E9, 9E9, 9E9]];
	VAR robtarget Openhole_6673 := [[397.66, -28.02, 177.07], [-0.134352, 0.694226, 0.681522, 0.18849], [0,0,0,0], [9E9, 9E9, 9E9, 9E9, 9E9, 9E9]];
	VAR robtarget Openhole_6674 := [[395.18, -28.08, 176.82], [-0.141049, 0.692896, 0.679728, 0.19486], [0,0,0,0], [9E9, 9E9, 9E9, 9E9, 9E9, 9E9]];
	VAR robtarget Openhole_6675 := [[394.33, -28.09, 176.74], [-0.143348, 0.692424, 0.679127, 0.196944], [0,0,0,0], [9E9, 9E9, 9E9, 9E9, 9E9, 9E9]];
	VAR robtarget Openhole_6676 := [[389.33, -28.09, 176.31], [-0.156675, 0.689531, 0.675558, 0.208856], [0,0,0,0], [9E9, 9E9, 9E9, 9E9, 9E9, 9E9]];
	VAR robtarget Openhole_6677 := [[362.33, -28.09, 176.39], [-0.183051, 0.683002, 0.683002, 0.183051], [0,0,0,0], [9E9, 9E9, 9E9, 9E9, 9E9, 9E9]];
	VAR robtarget Openhole_6678 := [[362.33, -27.21, 176.9], [-0.183051, 0.683002, 0.683002, 0.183051], [0,0,0,0], [9E9, 9E9, 9E9, 9E9, 9E9, 9E9]];
	VAR robtarget Openhole_6679 := [[374.33, -27.21, 176.86], [-0.183051, 0.683002, 0.683002, 0.183051], [0,0,0,0], [9E9, 9E9, 9E9, 9E9, 9E9, 9E9]];
	VAR robtarget Openhole_6680 := [[389.33, -27.21, 176.82], [-0.159203, 0.688952, 0.676318, 0.206384], [0,0,0,0], [9E9, 9E9, 9E9, 9E9, 9E9, 9E9]];
	VAR robtarget Openhole_6681 := [[394.26, -27.21, 177.21], [-0.146147, 0.691839, 0.679804, 0.194594], [0,0,0,0], [9E9, 9E9, 9E9, 9E9, 9E9, 9E9]];
	VAR robtarget Openhole_6682 := [[399.81, -27.04, 177.72], [-0.131284, 0.694813, 0.683774, 0.180148], [0,0,0,0], [9E9, 9E9, 9E9, 9E9, 9E9, 9E9]];
	VAR robtarget Openhole_6683 := [[400.3, -27.04, 177.76], [-0.12987, 0.695078, 0.684112, 0.178859], [0,0,0,0], [9E9, 9E9, 9E9, 9E9, 9E9, 9E9]];
	VAR robtarget Openhole_6684 := [[416.26, -27.54, 178.83], [-0.080359, 0.702526, 0.693876, 0.136147], [0,0,0,0], [9E9, 9E9, 9E9, 9E9, 9E9, 9E9]];
	VAR robtarget Openhole_6685 := [[416.76, -27.54, 178.87], [-0.078776, 0.702705, 0.694162, 0.134683], [0,0,0,0], [9E9, 9E9, 9E9, 9E9, 9E9, 9E9]];
	VAR robtarget Openhole_6686 := [[417.26, -27.54, 178.91], [-0.077202, 0.70288, 0.694448, 0.133202], [0,0,0,0], [9E9, 9E9, 9E9, 9E9, 9E9, 9E9]];
	VAR robtarget Openhole_6687 := [[422.73, -27.32, 179.42], [-0.060284, 0.704532, 0.697529, 0.115987], [0,0,0,0], [9E9, 9E9, 9E9, 9E9, 9E9, 9E9]];
	VAR robtarget Openhole_6688 := [[426.68, -26.85, 179.84], [-0.048887, 0.705415, 0.699689, 0.102154], [0,0,0,0], [9E9, 9E9, 9E9, 9E9, 9E9, 9E9]];
	VAR robtarget Openhole_6689 := [[430.07, -26.09, 180.23], [-0.040122, 0.705968, 0.701498, 0.088884], [0,0,0,0], [9E9, 9E9, 9E9, 9E9, 9E9, 9E9]];
	VAR robtarget Openhole_6690 := [[432.91, -25.19, 180.57], [-0.033638, 0.706306, 0.702934, 0.076708], [0,0,0,0], [9E9, 9E9, 9E9, 9E9, 9E9, 9E9]];
	VAR robtarget Openhole_6691 := [[433.37, -25.01, 180.62], [-0.03268, 0.706351, 0.70316, 0.074602], [0,0,0,0], [9E9, 9E9, 9E9, 9E9, 9E9, 9E9]];
	VAR robtarget Openhole_6692 := [[433.83, -24.82, 180.68], [-0.031768, 0.706393, 0.703383, 0.072471], [0,0,0,0], [9E9, 9E9, 9E9, 9E9, 9E9, 9E9]];
	VAR robtarget Openhole_6693 := [[434.29, -24.62, 180.73], [-0.030896, 0.706431, 0.703602, 0.07032], [0,0,0,0], [9E9, 9E9, 9E9, 9E9, 9E9, 9E9]];
	VAR robtarget Openhole_6694 := [[435.19, -24.2, 180.84], [-0.029269, 0.706501, 0.704024, 0.06596], [0,0,0,0], [9E9, 9E9, 9E9, 9E9, 9E9, 9E9]];
	VAR robtarget Openhole_6695 := [[436.52, -23.52, 180.99], [-0.027077, 0.706588, 0.704616, 0.059302], [0,0,0,0], [9E9, 9E9, 9E9, 9E9, 9E9, 9E9]];
	VAR robtarget Openhole_6696 := [[438.24, -22.52, 181.17], [-0.024642, 0.706677, 0.705321, 0.050225], [0,0,0,0], [9E9, 9E9, 9E9, 9E9, 9E9, 9E9]];
	VAR robtarget Openhole_6697 := [[440.79, -20.96, 181.38], [-0.021282, 0.706786, 0.706168, 0.036429], [0,0,0,0], [9E9, 9E9, 9E9, 9E9, 9E9, 9E9]];
	VAR robtarget Openhole_6698 := [[441.58, -20.63, 181.42], [-0.019713, 0.706832, 0.706352, 0.032657], [0,0,0,0], [9E9, 9E9, 9E9, 9E9, 9E9, 9E9]];
	VAR robtarget Openhole_6699 := [[443.72, -20.63, 181.45], [-0.012427, 0.706998, 0.706649, 0.025438], [0,0,0,0], [9E9, 9E9, 9E9, 9E9, 9E9, 9E9]];
	VAR robtarget Openhole_6700 := [[443.53, -19.52, 181.51], [-0.016872, 0.706905, 0.706754, 0.022334], [0,0,0,0], [9E9, 9E9, 9E9, 9E9, 9E9, 9E9]];
	VAR robtarget Openhole_6701 := [[441.39, -19.52, 181.5], [-0.024151, 0.706694, 0.706489, 0.029558], [0,0,0,0], [9E9, 9E9, 9E9, 9E9, 9E9, 9E9]];
	VAR robtarget Openhole_6702 := [[440.77, -19.7, 181.49], [-0.025645, 0.706642, 0.706373, 0.032213], [0,0,0,0], [9E9, 9E9, 9E9, 9E9, 9E9, 9E9]];
	VAR robtarget Openhole_6703 := [[440.32, -19.89, 181.47], [-0.026528, 0.706609, 0.706268, 0.034423], [0,0,0,0], [9E9, 9E9, 9E9, 9E9, 9E9, 9E9]];
	VAR robtarget Openhole_6704 := [[439.86, -20.1, 181.44], [-0.027351, 0.706578, 0.706156, 0.036653], [0,0,0,0], [9E9, 9E9, 9E9, 9E9, 9E9, 9E9]];
	VAR robtarget Openhole_6705 := [[439.41, -20.32, 181.42], [-0.028127, 0.706547, 0.706036, 0.038896], [0,0,0,0], [9E9, 9E9, 9E9, 9E9, 9E9, 9E9]];
	VAR robtarget Openhole_6706 := [[438.97, -20.55, 181.39], [-0.028829, 0.706519, 0.705908, 0.041161], [0,0,0,0], [9E9, 9E9, 9E9, 9E9, 9E9, 9E9]];
	VAR robtarget Openhole_6707 := [[438.54, -20.81, 181.36], [-0.029402, 0.706495, 0.70577, 0.043457], [0,0,0,0], [9E9, 9E9, 9E9, 9E9, 9E9, 9E9]];
	VAR robtarget Openhole_6708 := [[436.45, -22.16, 181.15], [-0.031894, 0.706387, 0.704967, 0.054968], [0,0,0,0], [9E9, 9E9, 9E9, 9E9, 9E9, 9E9]];
	VAR robtarget Openhole_6709 := [[436.02, -22.42, 181.11], [-0.032493, 0.70636, 0.704787, 0.057235], [0,0,0,0], [9E9, 9E9, 9E9, 9E9, 9E9, 9E9]];
	VAR robtarget Openhole_6710 := [[435.15, -22.9, 181.01], [-0.03381, 0.706298, 0.704408, 0.061724], [0,0,0,0], [9E9, 9E9, 9E9, 9E9, 9E9, 9E9]];
	VAR robtarget Openhole_6711 := [[434.26, -23.35, 180.91], [-0.035281, 0.706226, 0.704006, 0.066148], [0,0,0,0], [9E9, 9E9, 9E9, 9E9, 9E9, 9E9]];
	VAR robtarget Openhole_6712 := [[433.36, -23.77, 180.81], [-0.036891, 0.706144, 0.703583, 0.070507], [0,0,0,0], [9E9, 9E9, 9E9, 9E9, 9E9, 9E9]];
	VAR robtarget Openhole_6713 := [[432.44, -24.15, 180.71], [-0.038684, 0.706048, 0.703142, 0.074777], [0,0,0,0], [9E9, 9E9, 9E9, 9E9, 9E9, 9E9]];
	VAR robtarget Openhole_6714 := [[431.98, -24.33, 180.66], [-0.039644, 0.705995, 0.702915, 0.076877], [0,0,0,0], [9E9, 9E9, 9E9, 9E9, 9E9, 9E9]];
	VAR robtarget Openhole_6715 := [[431.04, -24.65, 180.55], [-0.041726, 0.705875, 0.702453, 0.080988], [0,0,0,0], [9E9, 9E9, 9E9, 9E9, 9E9, 9E9]];
	VAR robtarget Openhole_6716 := [[428.64, -25.31, 180.29], [-0.04747, 0.705512, 0.701241, 0.090888], [0,0,0,0], [9E9, 9E9, 9E9, 9E9, 9E9, 9E9]];
	VAR robtarget Openhole_6717 := [[426.69, -25.72, 180.08], [-0.052572, 0.70515, 0.700227, 0.098401], [0,0,0,0], [9E9, 9E9, 9E9, 9E9, 9E9, 9E9]];
	VAR robtarget Openhole_6718 := [[422.74, -26.21, 179.7], [-0.063892, 0.704214, 0.698127, 0.112333], [0,0,0,0], [9E9, 9E9, 9E9, 9E9, 9E9, 9E9]];
	VAR robtarget Openhole_6719 := [[417.77, -26.42, 179.3], [-0.079199, 0.702657, 0.695401, 0.12813], [0,0,0,0], [9E9, 9E9, 9E9, 9E9, 9E9, 9E9]];
	VAR robtarget Openhole_6720 := [[416.77, -26.42, 179.22], [-0.082341, 0.702296, 0.694845, 0.131115], [0,0,0,0], [9E9, 9E9, 9E9, 9E9, 9E9, 9E9]];
	VAR robtarget Openhole_6721 := [[416.27, -26.42, 179.19], [-0.083917, 0.70211, 0.694565, 0.132588], [0,0,0,0], [9E9, 9E9, 9E9, 9E9, 9E9, 9E9]];
	VAR robtarget Openhole_6722 := [[401.3, -26.08, 178.28], [-0.129942, 0.695065, 0.685515, 0.173404], [0,0,0,0], [9E9, 9E9, 9E9, 9E9, 9E9, 9E9]];
	VAR robtarget Openhole_6723 := [[400.8, -26.08, 178.25], [-0.131354, 0.694799, 0.685181, 0.174719], [0,0,0,0], [9E9, 9E9, 9E9, 9E9, 9E9, 9E9]];
	VAR robtarget Openhole_6724 := [[395.33, -26.26, 177.78], [-0.146039, 0.691862, 0.681319, 0.18922], [0,0,0,0], [9E9, 9E9, 9E9, 9E9, 9E9, 9E9]];
	VAR robtarget Openhole_6725 := [[394.83, -26.28, 177.73], [-0.147304, 0.691593, 0.680953, 0.190535], [0,0,0,0], [9E9, 9E9, 9E9, 9E9, 9E9, 9E9]];
	VAR robtarget Openhole_6726 := [[394.33, -26.32, 177.68], [-0.148543, 0.691328, 0.680573, 0.191888], [0,0,0,0], [9E9, 9E9, 9E9, 9E9, 9E9, 9E9]];
	VAR robtarget Openhole_6727 := [[394.33, -26.32, 177.68], [-0.148526, 0.691332, 0.680577, 0.191873], [0,0,0,0], [9E9, 9E9, 9E9, 9E9, 9E9, 9E9]];
	VAR robtarget Openhole_6728 := [[389.33, -26.32, 177.33], [-0.161727, 0.688364, 0.677068, 0.203911], [0,0,0,0], [9E9, 9E9, 9E9, 9E9, 9E9, 9E9]];
	VAR robtarget Openhole_6729 := [[362.33, -26.32, 177.41], [-0.183051, 0.683002, 0.683002, 0.183051], [0,0,0,0], [9E9, 9E9, 9E9, 9E9, 9E9, 9E9]];
	VAR robtarget Openhole_6730 := [[362.34, -24.22, 178.63], [-0.183051, 0.683002, 0.683002, 0.183051], [0,0,0,0], [9E9, 9E9, 9E9, 9E9, 9E9, 9E9]];
	VAR robtarget Openhole_6731 := [[389.34, -24.22, 178.54], [-0.167755, 0.686919, 0.678824, 0.197984], [0,0,0,0], [9E9, 9E9, 9E9, 9E9, 9E9, 9E9]];
	VAR robtarget Openhole_6732 := [[394.34, -24.22, 178.79], [-0.154705, 0.689976, 0.682261, 0.185795], [0,0,0,0], [9E9, 9E9, 9E9, 9E9, 9E9, 9E9]];
	VAR robtarget Openhole_6733 := [[395.31, -24.2, 178.85], [-0.152175, 0.690538, 0.682934, 0.183307], [0,0,0,0], [9E9, 9E9, 9E9, 9E9, 9E9, 9E9]];
	VAR robtarget Openhole_6734 := [[401.29, -23.97, 179.25], [-0.136374, 0.693832, 0.687063, 0.167165], [0,0,0,0], [9E9, 9E9, 9E9, 9E9, 9E9, 9E9]];
	VAR robtarget Openhole_6735 := [[403.29, -23.96, 179.35], [-0.130743, 0.694915, 0.688354, 0.161766], [0,0,0,0], [9E9, 9E9, 9E9, 9E9, 9E9, 9E9]];
	VAR robtarget Openhole_6736 := [[403.78, -23.96, 179.38], [-0.129311, 0.695183, 0.688671, 0.160413], [0,0,0,0], [9E9, 9E9, 9E9, 9E9, 9E9, 9E9]];
	VAR robtarget Openhole_6737 := [[416.77, -24.13, 179.94], [-0.089702, 0.701394, 0.696176, 0.123852], [0,0,0,0], [9E9, 9E9, 9E9, 9E9, 9E9, 9E9]];
	VAR robtarget Openhole_6738 := [[417.27, -24.13, 179.97], [-0.08814, 0.701592, 0.696441, 0.122351], [0,0,0,0], [9E9, 9E9, 9E9, 9E9, 9E9, 9E9]];
	VAR robtarget Openhole_6739 := [[422.76, -23.95, 180.28], [-0.071251, 0.703508, 0.699269, 0.104992], [0,0,0,0], [9E9, 9E9, 9E9, 9E9, 9E9, 9E9]];
	VAR robtarget Openhole_6740 := [[426.72, -23.49, 180.57], [-0.059869, 0.704568, 0.701222, 0.091036], [0,0,0,0], [9E9, 9E9, 9E9, 9E9, 9E9, 9E9]];
	VAR robtarget Openhole_6741 := [[427.7, -23.31, 180.65], [-0.057246, 0.704786, 0.701695, 0.087318], [0,0,0,0], [9E9, 9E9, 9E9, 9E9, 9E9, 9E9]];
	VAR robtarget Openhole_6742 := [[428.19, -23.21, 180.69], [-0.055977, 0.704888, 0.701928, 0.085421], [0,0,0,0], [9E9, 9E9, 9E9, 9E9, 9E9, 9E9]];
	VAR robtarget Openhole_6743 := [[430.12, -22.73, 180.86], [-0.05118, 0.705252, 0.702835, 0.077608], [0,0,0,0], [9E9, 9E9, 9E9, 9E9, 9E9, 9E9]];
	VAR robtarget Openhole_6744 := [[430.6, -22.59, 180.9], [-0.050053, 0.705333, 0.703054, 0.0756], [0,0,0,0], [9E9, 9E9, 9E9, 9E9, 9E9, 9E9]];
	VAR robtarget Openhole_6745 := [[432.02, -22.13, 181.02], [-0.046859, 0.705552, 0.703688, 0.069444], [0,0,0,0], [9E9, 9E9, 9E9, 9E9, 9E9, 9E9]];
	VAR robtarget Openhole_6746 := [[432.49, -21.97, 181.06], [-0.045848, 0.705619, 0.703891, 0.067356], [0,0,0,0], [9E9, 9E9, 9E9, 9E9, 9E9, 9E9]];
	VAR robtarget Openhole_6747 := [[433.88, -21.41, 181.19], [-0.043075, 0.705794, 0.704475, 0.060948], [0,0,0,0], [9E9, 9E9, 9E9, 9E9, 9E9, 9E9]];
	VAR robtarget Openhole_6748 := [[434.78, -20.99, 181.27], [-0.041473, 0.70589, 0.704841, 0.056557], [0,0,0,0], [9E9, 9E9, 9E9, 9E9, 9E9, 9E9]];
	VAR robtarget Openhole_6749 := [[435.23, -20.76, 181.31], [-0.040753, 0.705931, 0.705017, 0.054327], [0,0,0,0], [9E9, 9E9, 9E9, 9E9, 9E9, 9E9]];
	VAR robtarget Openhole_6750 := [[436.1, -20.28, 181.38], [-0.039455, 0.706005, 0.70535, 0.049814], [0,0,0,0], [9E9, 9E9, 9E9, 9E9, 9E9, 9E9]];
	VAR robtarget Openhole_6751 := [[436.54, -20.05, 181.42], [-0.038758, 0.706044, 0.705505, 0.047565], [0,0,0,0], [9E9, 9E9, 9E9, 9E9, 9E9, 9E9]];
	VAR robtarget Openhole_6752 := [[436.99, -19.83, 181.45], [-0.03797, 0.706087, 0.705652, 0.045343], [0,0,0,0], [9E9, 9E9, 9E9, 9E9, 9E9, 9E9]];
	VAR robtarget Openhole_6753 := [[437.9, -19.41, 181.5], [-0.036324, 0.706173, 0.705922, 0.040911], [0,0,0,0], [9E9, 9E9, 9E9, 9E9, 9E9, 9E9]];
	VAR robtarget Openhole_6754 := [[438.36, -19.23, 181.52], [-0.035373, 0.706221, 0.706045, 0.038741], [0,0,0,0], [9E9, 9E9, 9E9, 9E9, 9E9, 9E9]];
	VAR robtarget Openhole_6755 := [[438.84, -19.07, 181.54], [-0.034325, 0.706273, 0.706158, 0.036613], [0,0,0,0], [9E9, 9E9, 9E9, 9E9, 9E9, 9E9]];
	VAR robtarget Openhole_6756 := [[439.31, -18.93, 181.55], [-0.033201, 0.706327, 0.706264, 0.03452], [0,0,0,0], [9E9, 9E9, 9E9, 9E9, 9E9, 9E9]];
	VAR robtarget Openhole_6757 := [[440.28, -18.68, 181.57], [-0.030767, 0.706437, 0.706452, 0.030429], [0,0,0,0], [9E9, 9E9, 9E9, 9E9, 9E9, 9E9]];
	VAR robtarget Openhole_6758 := [[440.77, -18.58, 181.58], [-0.02943, 0.706494, 0.706534, 0.028454], [0,0,0,0], [9E9, 9E9, 9E9, 9E9, 9E9, 9E9]];
	VAR robtarget Openhole_6759 := [[441.27, -18.53, 181.58], [-0.027909, 0.706556, 0.706606, 0.026614], [0,0,0,0], [9E9, 9E9, 9E9, 9E9, 9E9, 9E9]];
	VAR robtarget Openhole_6760 := [[441.35, -18.53, 181.58], [-0.027644, 0.706566, 0.706615, 0.02636], [0,0,0,0], [9E9, 9E9, 9E9, 9E9, 9E9, 9E9]];
	VAR robtarget Openhole_6761 := [[443.12, -18.53, 181.57], [-0.021619, 0.706776, 0.706813, 0.020372], [0,0,0,0], [9E9, 9E9, 9E9, 9E9, 9E9, 9E9]];
	VAR robtarget Openhole_6762 := [[443.2, -17.55, 181.63], [-0.024694, 0.706675, 0.706908, 0.016763], [0,0,0,0], [9E9, 9E9, 9E9, 9E9, 9E9, 9E9]];
	VAR robtarget Openhole_6763 := [[441.43, -17.55, 181.65], [-0.030714, 0.706439, 0.706741, 0.022756], [0,0,0,0], [9E9, 9E9, 9E9, 9E9, 9E9, 9E9]];
	VAR robtarget Openhole_6764 := [[441.37, -17.54, 181.66], [-0.030961, 0.706429, 0.706735, 0.022941], [0,0,0,0], [9E9, 9E9, 9E9, 9E9, 9E9, 9E9]];
	VAR robtarget Openhole_6765 := [[440.87, -17.63, 181.66], [-0.032342, 0.706367, 0.706669, 0.024889], [0,0,0,0], [9E9, 9E9, 9E9, 9E9, 9E9, 9E9]];
	VAR robtarget Openhole_6766 := [[436.92, -18.24, 181.64], [-0.043587, 0.705762, 0.705962, 0.040226], [0,0,0,0], [9E9, 9E9, 9E9, 9E9, 9E9, 9E9]];
	VAR robtarget Openhole_6767 := [[436.43, -18.34, 181.63], [-0.044903, 0.70568, 0.705847, 0.04219], [0,0,0,0], [9E9, 9E9, 9E9, 9E9, 9E9, 9E9]];
	VAR robtarget Openhole_6768 := [[435.94, -18.42, 181.62], [-0.04629, 0.70559, 0.70573, 0.044102], [0,0,0,0], [9E9, 9E9, 9E9, 9E9, 9E9, 9E9]];
	VAR robtarget Openhole_6769 := [[434.95, -18.6, 181.6], [-0.048963, 0.70541, 0.705477, 0.047984], [0,0,0,0], [9E9, 9E9, 9E9, 9E9, 9E9, 9E9]];
	VAR robtarget Openhole_6770 := [[434.46, -18.67, 181.59], [-0.050369, 0.705311, 0.705346, 0.04987], [0,0,0,0], [9E9, 9E9, 9E9, 9E9, 9E9, 9E9]];
	VAR robtarget Openhole_6771 := [[433.97, -18.76, 181.58], [-0.051731, 0.705212, 0.705208, 0.051783], [0,0,0,0], [9E9, 9E9, 9E9, 9E9, 9E9, 9E9]];
	VAR robtarget Openhole_6772 := [[430.5, -19.24, 181.5], [-0.061593, 0.704419, 0.704132, 0.064797], [0,0,0,0], [9E9, 9E9, 9E9, 9E9, 9E9, 9E9]];
	VAR robtarget Openhole_6773 := [[429.51, -19.35, 181.48], [-0.064484, 0.70416, 0.70379, 0.06841], [0,0,0,0], [9E9, 9E9, 9E9, 9E9, 9E9, 9E9]];
	VAR robtarget Openhole_6774 := [[429.01, -19.4, 181.47], [-0.065961, 0.704024, 0.703615, 0.070183], [0,0,0,0], [9E9, 9E9, 9E9, 9E9, 9E9, 9E9]];
	VAR robtarget Openhole_6775 := [[424.02, -19.61, 181.4], [-0.081479, 0.702397, 0.701747, 0.086895], [0,0,0,0], [9E9, 9E9, 9E9, 9E9, 9E9, 9E9]];
	VAR robtarget Openhole_6776 := [[422.52, -19.62, 181.39], [-0.086259, 0.701826, 0.701142, 0.091649], [0,0,0,0], [9E9, 9E9, 9E9, 9E9, 9E9, 9E9]];
	VAR robtarget Openhole_6777 := [[422.02, -19.61, 181.39], [-0.087859, 0.701627, 0.700936, 0.09321], [0,0,0,0], [9E9, 9E9, 9E9, 9E9, 9E9, 9E9]];
	VAR robtarget Openhole_6778 := [[407.52, -19.42, 181.38], [-0.132576, 0.694567, 0.693879, 0.136134], [0,0,0,0], [9E9, 9E9, 9E9, 9E9, 9E9, 9E9]];
	VAR robtarget Openhole_6779 := [[407.02, -19.42, 181.38], [-0.13402, 0.69429, 0.693597, 0.137562], [0,0,0,0], [9E9, 9E9, 9E9, 9E9, 9E9, 9E9]];
	VAR robtarget Openhole_6780 := [[398.02, -19.61, 181.25], [-0.1585, 0.689114, 0.6881, 0.162843], [0,0,0,0], [9E9, 9E9, 9E9, 9E9, 9E9, 9E9]];
	VAR robtarget Openhole_6781 := [[394.35, -19.81, 181.13], [-0.167638, 0.686948, 0.68562, 0.172988], [0,0,0,0], [9E9, 9E9, 9E9, 9E9, 9E9, 9E9]];
	VAR robtarget Openhole_6782 := [[362.35, -19.81, 181.17], [-0.183051, 0.683002, 0.683002, 0.183051], [0,0,0,0], [9E9, 9E9, 9E9, 9E9, 9E9, 9E9]];
	VAR robtarget Openhole_6783 := [[362.35, -16.66, 182.99], [-0.183051, 0.683002, 0.683002, 0.183051], [0,0,0,0], [9E9, 9E9, 9E9, 9E9, 9E9, 9E9]];
	VAR robtarget Openhole_6784 := [[389.35, -16.66, 182.91], [-0.189336, 0.681287, 0.684715, 0.176538], [0,0,0,0], [9E9, 9E9, 9E9, 9E9, 9E9, 9E9]];
	VAR robtarget Openhole_6785 := [[394.35, -16.66, 182.79], [-0.176837, 0.684638, 0.687872, 0.163806], [0,0,0,0], [9E9, 9E9, 9E9, 9E9, 9E9, 9E9]];
	VAR robtarget Openhole_6786 := [[395.16, -16.63, 182.79], [-0.174857, 0.685146, 0.68839, 0.161614], [0,0,0,0], [9E9, 9E9, 9E9, 9E9, 9E9, 9E9]];
	VAR robtarget Openhole_6787 := [[403.65, -16.31, 182.73], [-0.153103, 0.690333, 0.693593, 0.13758], [0,0,0,0], [9E9, 9E9, 9E9, 9E9, 9E9, 9E9]];
	VAR robtarget Openhole_6788 := [[410.15, -16.25, 182.59], [-0.134864, 0.694126, 0.697085, 0.118627], [0,0,0,0], [9E9, 9E9, 9E9, 9E9, 9E9, 9E9]];
	VAR robtarget Openhole_6789 := [[410.65, -16.25, 182.58], [-0.133406, 0.694408, 0.697335, 0.11715], [0,0,0,0], [9E9, 9E9, 9E9, 9E9, 9E9, 9E9]];
	VAR robtarget Openhole_6790 := [[425.64, -16.49, 182.12], [-0.086572, 0.701787, 0.703485, 0.07148], [0,0,0,0], [9E9, 9E9, 9E9, 9E9, 9E9, 9E9]];
	VAR robtarget Openhole_6791 := [[437.63, -16.79, 181.79], [-0.046119, 0.705601, 0.706337, 0.032977], [0,0,0,0], [9E9, 9E9, 9E9, 9E9, 9E9, 9E9]];
	VAR robtarget Openhole_6792 := [[438.13, -16.79, 181.78], [-0.044449, 0.705708, 0.706414, 0.031291], [0,0,0,0], [9E9, 9E9, 9E9, 9E9, 9E9, 9E9]];
	VAR robtarget Openhole_6793 := [[438.63, -16.79, 181.77], [-0.042768, 0.705812, 0.706487, 0.029611], [0,0,0,0], [9E9, 9E9, 9E9, 9E9, 9E9, 9E9]];
	VAR robtarget Openhole_6794 := [[440.13, -16.73, 181.75], [-0.037909, 0.70609, 0.706687, 0.024376], [0,0,0,0], [9E9, 9E9, 9E9, 9E9, 9E9, 9E9]];
	VAR robtarget Openhole_6795 := [[440.63, -16.69, 181.74], [-0.036359, 0.706171, 0.706747, 0.022563], [0,0,0,0], [9E9, 9E9, 9E9, 9E9, 9E9, 9E9]];
	VAR robtarget Openhole_6796 := [[441.11, -16.58, 181.74], [-0.03509, 0.706236, 0.706808, 0.020541], [0,0,0,0], [9E9, 9E9, 9E9, 9E9, 9E9, 9E9]];
	VAR robtarget Openhole_6797 := [[441.66, -16.48, 181.73], [-0.03356, 0.70631, 0.706868, 0.018373], [0,0,0,0], [9E9, 9E9, 9E9, 9E9, 9E9, 9E9]];
	VAR robtarget Openhole_6798 := [[443.56, -16.48, 181.68], [-0.027128, 0.706586, 0.707006, 0.011959], [0,0,0,0], [9E9, 9E9, 9E9, 9E9, 9E9, 9E9]];
	VAR robtarget Openhole_6799 := [[443.93, -15.46, 181.73], [-0.029352, 0.706497, 0.70707, 0.007216], [0,0,0,0], [9E9, 9E9, 9E9, 9E9, 9E9, 9E9]];
	VAR robtarget Openhole_6800 := [[442.03, -15.46, 181.79], [-0.035783, 0.706201, 0.706975, 0.013637], [0,0,0,0], [9E9, 9E9, 9E9, 9E9, 9E9, 9E9]];
	VAR robtarget Openhole_6801 := [[441.46, -15.51, 181.81], [-0.037542, 0.706109, 0.706931, 0.015744], [0,0,0,0], [9E9, 9E9, 9E9, 9E9, 9E9, 9E9]];
	VAR robtarget Openhole_6802 := [[440.97, -15.59, 181.82], [-0.038914, 0.706035, 0.706885, 0.017699], [0,0,0,0], [9E9, 9E9, 9E9, 9E9, 9E9, 9E9]];
	VAR robtarget Openhole_6803 := [[439.97, -15.62, 181.85], [-0.042187, 0.705847, 0.70679, 0.02117], [0,0,0,0], [9E9, 9E9, 9E9, 9E9, 9E9, 9E9]];
	VAR robtarget Openhole_6804 := [[439.47, -15.62, 181.87], [-0.043884, 0.705744, 0.706738, 0.022842], [0,0,0,0], [9E9, 9E9, 9E9, 9E9, 9E9, 9E9]];
	VAR robtarget Openhole_6805 := [[438.97, -15.61, 181.88], [-0.045615, 0.705634, 0.706683, 0.024474], [0,0,0,0], [9E9, 9E9, 9E9, 9E9, 9E9, 9E9]];
	VAR robtarget Openhole_6806 := [[438.47, -15.58, 181.9], [-0.047379, 0.705518, 0.706626, 0.026068], [0,0,0,0], [9E9, 9E9, 9E9, 9E9, 9E9, 9E9]];
	VAR robtarget Openhole_6807 := [[437.48, -15.49, 181.95], [-0.05101, 0.705264, 0.706507, 0.029121], [0,0,0,0], [9E9, 9E9, 9E9, 9E9, 9E9, 9E9]];
	VAR robtarget Openhole_6808 := [[431.51, -14.94, 182.24], [-0.072676, 0.703362, 0.705534, 0.047142], [0,0,0,0], [9E9, 9E9, 9E9, 9E9, 9E9, 9E9]];
	VAR robtarget Openhole_6809 := [[422.53, -14.66, 182.67], [-0.10246, 0.699644, 0.703069, 0.075456], [0,0,0,0], [9E9, 9E9, 9E9, 9E9, 9E9, 9E9]];
	VAR robtarget Openhole_6810 := [[413.54, -14.6, 183.07], [-0.130108, 0.695034, 0.699523, 0.103285], [0,0,0,0], [9E9, 9E9, 9E9, 9E9, 9E9, 9E9]];
	VAR robtarget Openhole_6811 := [[413.04, -14.6, 183.09], [-0.131583, 0.694756, 0.699297, 0.104802], [0,0,0,0], [9E9, 9E9, 9E9, 9E9, 9E9, 9E9]];
	VAR robtarget Openhole_6812 := [[401.55, -14.77, 183.5], [-0.163536, 0.687936, 0.693352, 0.13879], [0,0,0,0], [9E9, 9E9, 9E9, 9E9, 9E9, 9E9]];
	VAR robtarget Openhole_6813 := [[394.35, -15.07, 183.63], [-0.181459, 0.683427, 0.688959, 0.159169], [0,0,0,0], [9E9, 9E9, 9E9, 9E9, 9E9, 9E9]];
	VAR robtarget Openhole_6814 := [[389.35, -15.07, 183.82], [-0.193842, 0.680019, 0.685865, 0.172014], [0,0,0,0], [9E9, 9E9, 9E9, 9E9, 9E9, 9E9]];
	VAR robtarget Openhole_6815 := [[362.35, -15.07, 183.91], [-0.183051, 0.683002, 0.683002, 0.183051], [0,0,0,0], [9E9, 9E9, 9E9, 9E9, 9E9, 9E9]];
	VAR robtarget Openhole_6816 := [[362.36, -14.11, 184.47], [-0.183051, 0.683002, 0.683002, 0.183051], [0,0,0,0], [9E9, 9E9, 9E9, 9E9, 9E9, 9E9]];
	VAR robtarget Openhole_6817 := [[389.36, -14.11, 184.38], [-0.196576, 0.679233, 0.68655, 0.169262], [0,0,0,0], [9E9, 9E9, 9E9, 9E9, 9E9, 9E9]];
	VAR robtarget Openhole_6818 := [[394.35, -14.11, 184.14], [-0.184264, 0.682676, 0.689605, 0.156348], [0,0,0,0], [9E9, 9E9, 9E9, 9E9, 9E9, 9E9]];
	VAR robtarget Openhole_6819 := [[404.57, -13.71, 183.83], [-0.158487, 0.689117, 0.695604, 0.127026], [0,0,0,0], [9E9, 9E9, 9E9, 9E9, 9E9, 9E9]];
	VAR robtarget Openhole_6820 := [[419.55, -13.55, 183.11], [-0.115314, 0.697641, 0.702419, 0.081284], [0,0,0,0], [9E9, 9E9, 9E9, 9E9, 9E9, 9E9]];
	VAR robtarget Openhole_6821 := [[420.05, -13.55, 183.09], [-0.113777, 0.697893, 0.7026, 0.079707], [0,0,0,0], [9E9, 9E9, 9E9, 9E9, 9E9, 9E9]];
	VAR robtarget Openhole_6822 := [[430.53, -13.69, 182.51], [-0.080025, 0.702564, 0.705594, 0.046234], [0,0,0,0], [9E9, 9E9, 9E9, 9E9, 9E9, 9E9]];
	VAR robtarget Openhole_6823 := [[435.51, -14.05, 182.2], [-0.062452, 0.704344, 0.706433, 0.030854], [0,0,0,0], [9E9, 9E9, 9E9, 9E9, 9E9, 9E9]];
	VAR robtarget Openhole_6824 := [[438.48, -14.4, 182.02], [-0.051315, 0.705242, 0.706762, 0.022071], [0,0,0,0], [9E9, 9E9, 9E9, 9E9, 9E9, 9E9]];
	VAR robtarget Openhole_6825 := [[438.98, -14.45, 182], [-0.049499, 0.705372, 0.706808, 0.020539], [0,0,0,0], [9E9, 9E9, 9E9, 9E9, 9E9, 9E9]];
	VAR robtarget Openhole_6826 := [[439.48, -14.47, 181.97], [-0.047733, 0.705494, 0.706853, 0.018947], [0,0,0,0], [9E9, 9E9, 9E9, 9E9, 9E9, 9E9]];
	VAR robtarget Openhole_6827 := [[439.98, -14.49, 181.95], [-0.046015, 0.705608, 0.706895, 0.017298], [0,0,0,0], [9E9, 9E9, 9E9, 9E9, 9E9, 9E9]];
	VAR robtarget Openhole_6828 := [[440.98, -14.49, 181.91], [-0.04263, 0.705821, 0.706969, 0.01394], [0,0,0,0], [9E9, 9E9, 9E9, 9E9, 9E9, 9E9]];
	VAR robtarget Openhole_6829 := [[441.98, -14.53, 181.86], [-0.039116, 0.706024, 0.707026, 0.010705], [0,0,0,0], [9E9, 9E9, 9E9, 9E9, 9E9, 9E9]];
	VAR robtarget Openhole_6830 := [[442.51, -14.54, 181.84], [-0.037266, 0.706124, 0.70705, 0.008939], [0,0,0,0], [9E9, 9E9, 9E9, 9E9, 9E9, 9E9]];
	VAR robtarget Openhole_6831 := [[444.29, -14.54, 181.76], [-0.03125, 0.706416, 0.707101, 0.002927], [0,0,0,0], [9E9, 9E9, 9E9, 9E9, 9E9, 9E9]];
	VAR robtarget Openhole_6832 := [[445.21, -13.31, 181.77], [-0.032306, 0.706368, 0.707093, -0.004384], [0,0,0,0], [9E9, 9E9, 9E9, 9E9, 9E9, 9E9]];
	VAR robtarget Openhole_6833 := [[443.44, -13.31, 181.87], [-0.038325, 0.706067, 0.707105, 0.001635], [0,0,0,0], [9E9, 9E9, 9E9, 9E9, 9E9, 9E9]];
	VAR robtarget Openhole_6834 := [[442.75, -13.1, 181.92], [-0.041365, 0.705896, 0.707099, 0.003278], [0,0,0,0], [9E9, 9E9, 9E9, 9E9, 9E9, 9E9]];
	VAR robtarget Openhole_6835 := [[440.25, -13.05, 182.07], [-0.049979, 0.705338, 0.707013, 0.011532], [0,0,0,0], [9E9, 9E9, 9E9, 9E9, 9E9, 9E9]];
	VAR robtarget Openhole_6836 := [[433.78, -12.57, 182.51], [-0.073116, 0.703316, 0.706396, 0.031703], [0,0,0,0], [9E9, 9E9, 9E9, 9E9, 9E9, 9E9]];
	VAR robtarget Openhole_6837 := [[427.8, -12.45, 182.9], [-0.092976, 0.700968, 0.705254, 0.051148], [0,0,0,0], [9E9, 9E9, 9E9, 9E9, 9E9, 9E9]];
	VAR robtarget Openhole_6838 := [[427.3, -12.45, 182.94], [-0.094574, 0.700754, 0.705134, 0.052785], [0,0,0,0], [9E9, 9E9, 9E9, 9E9, 9E9, 9E9]];
	VAR robtarget Openhole_6839 := [[408.83, -12.69, 184.01], [-0.149733, 0.691072, 0.698273, 0.111421], [0,0,0,0], [9E9, 9E9, 9E9, 9E9, 9E9, 9E9]];
	VAR robtarget Openhole_6840 := [[397.35, -13.06, 184.53], [-0.179687, 0.683895, 0.692029, 0.145246], [0,0,0,0], [9E9, 9E9, 9E9, 9E9, 9E9, 9E9]];
	VAR robtarget Openhole_6841 := [[394.34, -13.23, 184.61], [-0.186879, 0.681965, 0.690173, 0.153822], [0,0,0,0], [9E9, 9E9, 9E9, 9E9, 9E9, 9E9]];
	VAR robtarget Openhole_6842 := [[389.36, -13.23, 184.89], [-0.199074, 0.678505, 0.687166, 0.166742], [0,0,0,0], [9E9, 9E9, 9E9, 9E9, 9E9, 9E9]];
	VAR robtarget Openhole_6843 := [[362.36, -13.23, 184.98], [-0.183051, 0.683002, 0.683002, 0.183051], [0,0,0,0], [9E9, 9E9, 9E9, 9E9, 9E9, 9E9]];
	VAR robtarget Openhole_6844 := [[362.36, -12.34, 185.49], [-0.183051, 0.683002, 0.683002, 0.183051], [0,0,0,0], [9E9, 9E9, 9E9, 9E9, 9E9, 9E9]];
	VAR robtarget Openhole_6845 := [[374.36, -12.34, 185.45], [-0.183051, 0.683002, 0.683002, 0.183051], [0,0,0,0], [9E9, 9E9, 9E9, 9E9, 9E9, 9E9]];
	VAR robtarget Openhole_6846 := [[389.36, -12.34, 185.4], [-0.201568, 0.677769, 0.687773, 0.16422], [0,0,0,0], [9E9, 9E9, 9E9, 9E9, 9E9, 9E9]];
	VAR robtarget Openhole_6847 := [[394.34, -12.34, 185.08], [-0.189433, 0.68126, 0.690745, 0.151233], [0,0,0,0], [9E9, 9E9, 9E9, 9E9, 9E9, 9E9]];
	VAR robtarget Openhole_6848 := [[404.84, -11.88, 184.6], [-0.163337, 0.687983, 0.696736, 0.120661], [0,0,0,0], [9E9, 9E9, 9E9, 9E9, 9E9, 9E9]];
	VAR robtarget Openhole_6849 := [[429.78, -11.27, 183], [-0.090529, 0.701288, 0.705934, 0.040701], [0,0,0,0], [9E9, 9E9, 9E9, 9E9, 9E9, 9E9]];
	VAR robtarget Openhole_6850 := [[431.77, -11.25, 182.86], [-0.084111, 0.702086, 0.706288, 0.034022], [0,0,0,0], [9E9, 9E9, 9E9, 9E9, 9E9, 9E9]];
	VAR robtarget Openhole_6851 := [[432.27, -11.25, 182.82], [-0.082483, 0.70228, 0.706366, 0.032361], [0,0,0,0], [9E9, 9E9, 9E9, 9E9, 9E9, 9E9]];
	VAR robtarget Openhole_6852 := [[441.74, -11.43, 182.1], [-0.050437, 0.705306, 0.707106, 0.001026], [0,0,0,0], [9E9, 9E9, 9E9, 9E9, 9E9, 9E9]];
	VAR robtarget Openhole_6853 := [[442.24, -11.45, 182.06], [-0.048669, 0.70543, 0.707107, -0.000574], [0,0,0,0], [9E9, 9E9, 9E9, 9E9, 9E9, 9E9]];
	VAR robtarget Openhole_6854 := [[443.23, -11.52, 181.98], [-0.045065, 0.705669, 0.707097, -0.003706], [0,0,0,0], [9E9, 9E9, 9E9, 9E9, 9E9, 9E9]];
	VAR robtarget Openhole_6855 := [[444.23, -11.62, 181.91], [-0.041372, 0.705895, 0.707075, -0.006743], [0,0,0,0], [9E9, 9E9, 9E9, 9E9, 9E9, 9E9]];
	VAR robtarget Openhole_6856 := [[444.72, -11.69, 181.87], [-0.039482, 0.706004, 0.707059, -0.00821], [0,0,0,0], [9E9, 9E9, 9E9, 9E9, 9E9, 9E9]];
	VAR robtarget Openhole_6857 := [[445.25, -11.83, 181.83], [-0.037191, 0.706128, 0.707042, -0.009548], [0,0,0,0], [9E9, 9E9, 9E9, 9E9, 9E9, 9E9]];
	VAR robtarget Openhole_6858 := [[454.83, -12.87, 181.22], [-0.001006, 0.707106, 0.70606, -0.038453], [0,0,0,0], [9E9, 9E9, 9E9, 9E9, 9E9, 9E9]];
	VAR robtarget Openhole_6859 := [[455.36, -12.53, 181.17], [-0.000348, 0.707107, 0.705895, -0.041387], [0,0,0,0], [9E9, 9E9, 9E9, 9E9, 9E9, 9E9]];
	VAR robtarget Openhole_6860 := [[455.8, -12.3, 181.12], [0.000393, 0.707107, 0.705759, -0.043645], [0,0,0,0], [9E9, 9E9, 9E9, 9E9, 9E9, 9E9]];
	VAR robtarget Openhole_6861 := [[456.25, -12.09, 181.08], [0.001208, 0.707106, 0.705617, -0.045876], [0,0,0,0], [9E9, 9E9, 9E9, 9E9, 9E9, 9E9]];
	VAR robtarget Openhole_6862 := [[456.7, -11.89, 181.04], [0.002062, 0.707104, 0.70547, -0.048088], [0,0,0,0], [9E9, 9E9, 9E9, 9E9, 9E9, 9E9]];
	VAR robtarget Openhole_6863 := [[457.17, -11.7, 180.99], [0.003025, 0.7071, 0.705319, -0.050254], [0,0,0,0], [9E9, 9E9, 9E9, 9E9, 9E9, 9E9]];
	VAR robtarget Openhole_6864 := [[458.11, -11.38, 180.9], [0.005123, 0.707088, 0.705003, -0.0545], [0,0,0,0], [9E9, 9E9, 9E9, 9E9, 9E9, 9E9]];
	VAR robtarget Openhole_6865 := [[464.3, -9.52, 180.17], [0.019895, 0.706827, 0.702436, -0.081137], [0,0,0,0], [9E9, 9E9, 9E9, 9E9, 9E9, 9E9]];
	VAR robtarget Openhole_6866 := [[464.77, -9.39, 180.11], [0.02107, 0.706793, 0.702203, -0.083134], [0,0,0,0], [9E9, 9E9, 9E9, 9E9, 9E9, 9E9]];
	VAR robtarget Openhole_6867 := [[469.61, -8.3, 179.45], [0.03368, 0.706304, 0.69967, -0.102286], [0,0,0,0], [9E9, 9E9, 9E9, 9E9, 9E9, 9E9]];
	VAR robtarget Openhole_6868 := [[474.02, -7.68, 178.85], [0.046276, 0.705591, 0.697163, -0.118169], [0,0,0,0], [9E9, 9E9, 9E9, 9E9, 9E9, 9E9]];
	VAR robtarget Openhole_6869 := [[478.47, -7.38, 178.28], [0.059876, 0.704567, 0.694543, -0.132702], [0,0,0,0], [9E9, 9E9, 9E9, 9E9, 9E9, 9E9]];
	VAR robtarget Openhole_6870 := [[480.96, -7.35, 177.99], [0.06777, 0.703852, 0.693067, -0.140205], [0,0,0,0], [9E9, 9E9, 9E9, 9E9, 9E9, 9E9]];
	VAR robtarget Openhole_6871 := [[481.45, -7.35, 177.93], [0.069362, 0.703697, 0.69277, -0.141668], [0,0,0,0], [9E9, 9E9, 9E9, 9E9, 9E9, 9E9]];
	VAR robtarget Openhole_6872 := [[487.92, -7.59, 177.3], [0.090383, 0.701307, 0.688878, -0.159523], [0,0,0,0], [9E9, 9E9, 9E9, 9E9, 9E9, 9E9]];
	VAR robtarget Openhole_6873 := [[499.86, -8.3, 176.33], [0.127809, 0.69546, 0.681292, -0.189317], [0,0,0,0], [9E9, 9E9, 9E9, 9E9, 9E9, 9E9]];
	VAR robtarget Openhole_6874 := [[501.35, -8.33, 176.18], [0.132072, 0.694663, 0.680255, -0.193009], [0,0,0,0], [9E9, 9E9, 9E9, 9E9, 9E9, 9E9]];
	VAR robtarget Openhole_6875 := [[501.85, -8.33, 176.13], [0.133456, 0.694399, 0.679901, -0.194253], [0,0,0,0], [9E9, 9E9, 9E9, 9E9, 9E9, 9E9]];
	VAR robtarget Openhole_6876 := [[503.83, -8.3, 175.92], [0.138865, 0.693337, 0.678459, -0.199231], [0,0,0,0], [9E9, 9E9, 9E9, 9E9, 9E9, 9E9]];
	VAR robtarget Openhole_6877 := [[504.35, -8.28, 175.85], [0.140205, 0.693067, 0.678062, -0.200578], [0,0,0,0], [9E9, 9E9, 9E9, 9E9, 9E9, 9E9]];
	VAR robtarget Openhole_6878 := [[509.33, -8.28, 175.33], [0.183051, 0.683002, 0.683002, -0.183051], [0,0,0,0], [9E9, 9E9, 9E9, 9E9, 9E9, 9E9]];
	VAR robtarget Openhole_6879 := [[536.33, -8.27, 175.25], [0.183051, 0.683002, 0.683002, -0.183051], [0,0,0,0], [9E9, 9E9, 9E9, 9E9, 9E9, 9E9]];
	VAR robtarget Openhole_6880 := [[536.33, -9.15, 175.75], [0.183051, 0.683002, 0.683002, -0.183051], [0,0,0,0], [9E9, 9E9, 9E9, 9E9, 9E9, 9E9]];
	VAR robtarget Openhole_6881 := [[509.33, -9.15, 175.84], [0.183051, 0.683002, 0.683002, -0.183051], [0,0,0,0], [9E9, 9E9, 9E9, 9E9, 9E9, 9E9]];
	VAR robtarget Openhole_6882 := [[504.33, -9.15, 176.31], [0.142686, 0.692561, 0.678811, -0.19803], [0,0,0,0], [9E9, 9E9, 9E9, 9E9, 9E9, 9E9]];
	VAR robtarget Openhole_6883 := [[503.69, -9.17, 176.39], [0.141021, 0.692902, 0.67929, -0.196381], [0,0,0,0], [9E9, 9E9, 9E9, 9E9, 9E9, 9E9]];
	VAR robtarget Openhole_6884 := [[503.19, -9.2, 176.45], [0.139765, 0.693156, 0.679668, -0.195067], [0,0,0,0], [9E9, 9E9, 9E9, 9E9, 9E9, 9E9]];
	VAR robtarget Openhole_6885 := [[500.21, -9.26, 176.76], [0.13167, 0.69474, 0.681817, -0.187419], [0,0,0,0], [9E9, 9E9, 9E9, 9E9, 9E9, 9E9]];
	VAR robtarget Openhole_6886 := [[499.71, -9.26, 176.8], [0.130265, 0.695004, 0.682162, -0.186157], [0,0,0,0], [9E9, 9E9, 9E9, 9E9, 9E9, 9E9]];
	VAR robtarget Openhole_6887 := [[491.74, -8.94, 177.42], [0.106193, 0.699087, 0.687343, -0.166009], [0,0,0,0], [9E9, 9E9, 9E9, 9E9, 9E9, 9E9]];
	VAR robtarget Openhole_6888 := [[482.78, -8.57, 178.17], [0.077474, 0.70285, 0.692751, -0.141761], [0,0,0,0], [9E9, 9E9, 9E9, 9E9, 9E9, 9E9]];
	VAR robtarget Openhole_6889 := [[481.79, -8.56, 178.27], [0.074304, 0.703192, 0.69334, -0.138853], [0,0,0,0], [9E9, 9E9, 9E9, 9E9, 9E9, 9E9]];
	VAR robtarget Openhole_6890 := [[481.29, -8.56, 178.32], [0.072727, 0.703357, 0.693633, -0.137379], [0,0,0,0], [9E9, 9E9, 9E9, 9E9, 9E9, 9E9]];
	VAR robtarget Openhole_6891 := [[476.33, -8.73, 178.87], [0.057274, 0.704783, 0.696524, -0.121877], [0,0,0,0], [9E9, 9E9, 9E9, 9E9, 9E9, 9E9]];
	VAR robtarget Openhole_6892 := [[471.89, -9.23, 179.42], [0.044349, 0.705715, 0.699045, -0.106471], [0,0,0,0], [9E9, 9E9, 9E9, 9E9, 9E9, 9E9]];
	VAR robtarget Openhole_6893 := [[468.97, -9.8, 179.8], [0.036516, 0.706163, 0.700649, -0.095347], [0,0,0,0], [9E9, 9E9, 9E9, 9E9, 9E9, 9E9]];
	VAR robtarget Openhole_6894 := [[466.57, -10.43, 180.12], [0.030572, 0.706446, 0.701912, -0.085555], [0,0,0,0], [9E9, 9E9, 9E9, 9E9, 9E9, 9E9]];
	VAR robtarget Openhole_6895 := [[463.74, -11.36, 180.48], [0.024207, 0.706692, 0.703305, -0.073222], [0,0,0,0], [9E9, 9E9, 9E9, 9E9, 9E9, 9E9]];
	VAR robtarget Openhole_6896 := [[461.9, -12.1, 180.7], [0.020458, 0.706811, 0.704143, -0.064677], [0,0,0,0], [9E9, 9E9, 9E9, 9E9, 9E9, 9E9]];
	VAR robtarget Openhole_6897 := [[460.54, -12.71, 180.86], [0.017883, 0.706881, 0.704714, -0.058126], [0,0,0,0], [9E9, 9E9, 9E9, 9E9, 9E9, 9E9]];
	VAR robtarget Openhole_6898 := [[459.64, -13.14, 180.96], [0.016317, 0.706918, 0.705066, -0.053685], [0,0,0,0], [9E9, 9E9, 9E9, 9E9, 9E9, 9E9]];
	VAR robtarget Openhole_6899 := [[459.2, -13.37, 181.01], [0.015593, 0.706935, 0.705233, -0.05144], [0,0,0,0], [9E9, 9E9, 9E9, 9E9, 9E9, 9E9]];
	VAR robtarget Openhole_6900 := [[458.76, -13.61, 181.05], [0.014915, 0.706949, 0.705395, -0.049177], [0,0,0,0], [9E9, 9E9, 9E9, 9E9, 9E9, 9E9]];
	VAR robtarget Openhole_6901 := [[457.91, -14.13, 181.14], [0.013757, 0.706973, 0.7057, -0.044588], [0,0,0,0], [9E9, 9E9, 9E9, 9E9, 9E9, 9E9]];
